    	END_IF;
    END_WHILE;
END_IF;
(* Rung 3 *)
IF P_On THEN AryByteTo(In := OUT[1], Size := 300, Order := _HIGH_LOW, OutVal := GBWORD); END_IF;
(* Rung 4 *)
IF P_On THEN
    unicode[0]:=16#4e00;
    unicode[1]:=16#4e01;
    unicode[2]:=16#4e03;
    unicode[3]:=16#4e07;
    unicode[4]:=16#4e08;
    unicode[5]:=16#4e09;
    unicode[6]:=16#4e0a;
    unicode[7]:=16#4e0b;
    unicode[8]:=16#4e0c;
    unicode[9]:=16#4e0d;
    unicode[10]:=16#4e0e;
    unicode[11]:=16#4e10;
    unicode[12]:=16#4e11;
    unicode[13]:=16#4e13;
    unicode[14]:=16#4e14;
    unicode[15]:=16#4e15;
    unicode[16]:=16#4e16;
    unicode[17]:=16#4e18;
    unicode[18]:=16#4e19;
    unicode[19]:=16#4e1a;
    unicode[20]:=16#4e1b;
    unicode[21]:=16#4e1c;
    unicode[22]:=16#4e1d;
    unicode[23]:=16#4e1e;
    unicode[24]:=16#4e22;
    unicode[25]:=16#4e24;
    unicode[26]:=16#4e25;
    unicode[27]:=16#4e27;
    unicode[28]:=16#4e28;
    unicode[29]:=16#4e2a;
    unicode[30]:=16#4e2b;
    unicode[31]:=16#4e2c;
    unicode[32]:=16#4e2d;
    unicode[33]:=16#4e30;
    unicode[34]:=16#4e32;
    unicode[35]:=16#4e34;
    unicode[36]:=16#4e36;
    unicode[37]:=16#4e38;
    unicode[38]:=16#4e39;
    unicode[39]:=16#4e3a;
    unicode[40]:=16#4e3b;
    unicode[41]:=16#4e3d;
    unicode[42]:=16#4e3e;
    unicode[43]:=16#4e3f;
    unicode[44]:=16#4e43;
    unicode[45]:=16#4e45;
    unicode[46]:=16#4e47;
    unicode[47]:=16#4e48;
    unicode[48]:=16#4e49;
    unicode[49]:=16#4e4b;
    unicode[50]:=16#4e4c;
    unicode[51]:=16#4e4d;
    unicode[52]:=16#4e4e;
    unicode[53]:=16#4e4f;
    unicode[54]:=16#4e50;
    unicode[55]:=16#4e52;
    unicode[56]:=16#4e53;
    unicode[57]:=16#4e54;
    unicode[58]:=16#4e56;
    unicode[59]:=16#4e58;
    unicode[60]:=16#4e59;
    unicode[61]:=16#4e5c;
    unicode[62]:=16#4e5d;
    unicode[63]:=16#4e5e;
    unicode[64]:=16#4e5f;
    unicode[65]:=16#4e60;
    unicode[66]:=16#4e61;
    unicode[67]:=16#4e66;
    unicode[68]:=16#4e69;
    unicode[69]:=16#4e70;
    unicode[70]:=16#4e71;
    unicode[71]:=16#4e73;
    unicode[72]:=16#4e7e;
    unicode[73]:=16#4e86;
    unicode[74]:=16#4e88;
    unicode[75]:=16#4e89;
    unicode[76]:=16#4e8b;
    unicode[77]:=16#4e8c;
    unicode[78]:=16#4e8d;
    unicode[79]:=16#4e8e;
    unicode[80]:=16#4e8f;
    unicode[81]:=16#4e91;
    unicode[82]:=16#4e92;
    unicode[83]:=16#4e93;
    unicode[84]:=16#4e94;
    unicode[85]:=16#4e95;
    unicode[86]:=16#4e98;
    unicode[87]:=16#4e9a;
    unicode[88]:=16#4e9b;
    unicode[89]:=16#4e9f;
    unicode[90]:=16#4ea0;
    unicode[91]:=16#4ea1;
    unicode[92]:=16#4ea2;
    unicode[93]:=16#4ea4;
    unicode[94]:=16#4ea5;
    unicode[95]:=16#4ea6;
    unicode[96]:=16#4ea7;
    unicode[97]:=16#4ea8;
    unicode[98]:=16#4ea9;
    unicode[99]:=16#4eab;
    unicode[100]:=16#4eac;
    unicode[101]:=16#4ead;
    unicode[102]:=16#4eae;
    unicode[103]:=16#4eb2;
    unicode[104]:=16#4eb3;
    unicode[105]:=16#4eb5;
    unicode[106]:=16#4eba;
    unicode[107]:=16#4ebb;
    unicode[108]:=16#4ebf;
    unicode[109]:=16#4ec0;
    unicode[110]:=16#4ec1;
    unicode[111]:=16#4ec2;
    unicode[112]:=16#4ec3;
    unicode[113]:=16#4ec4;
    unicode[114]:=16#4ec5;
    unicode[115]:=16#4ec6;
    unicode[116]:=16#4ec7;
    unicode[117]:=16#4ec9;
    unicode[118]:=16#4eca;
    unicode[119]:=16#4ecb;
    unicode[120]:=16#4ecd;
    unicode[121]:=16#4ece;
    unicode[122]:=16#4ed1;
    unicode[123]:=16#4ed3;
    unicode[124]:=16#4ed4;
    unicode[125]:=16#4ed5;
    unicode[126]:=16#4ed6;
    unicode[127]:=16#4ed7;
    unicode[128]:=16#4ed8;
    unicode[129]:=16#4ed9;
    unicode[130]:=16#4edd;
    unicode[131]:=16#4ede;
    unicode[132]:=16#4edf;
    unicode[133]:=16#4ee1;
    unicode[134]:=16#4ee3;
    unicode[135]:=16#4ee4;
    unicode[136]:=16#4ee5;
    unicode[137]:=16#4ee8;
    unicode[138]:=16#4eea;
    unicode[139]:=16#4eeb;
    unicode[140]:=16#4eec;
    unicode[141]:=16#4ef0;
    unicode[142]:=16#4ef2;
    unicode[143]:=16#4ef3;
    unicode[144]:=16#4ef5;
    unicode[145]:=16#4ef6;
    unicode[146]:=16#4ef7;
    unicode[147]:=16#4efb;
    unicode[148]:=16#4efd;
    unicode[149]:=16#4eff;
    unicode[150]:=16#4f01;
    unicode[151]:=16#4f09;
    unicode[152]:=16#4f0a;
    unicode[153]:=16#4f0d;
    unicode[154]:=16#4f0e;
    unicode[155]:=16#4f0f;
    unicode[156]:=16#4f10;
    unicode[157]:=16#4f11;
    unicode[158]:=16#4f17;
    unicode[159]:=16#4f18;
    unicode[160]:=16#4f19;
    unicode[161]:=16#4f1a;
    unicode[162]:=16#4f1b;
    unicode[163]:=16#4f1e;
    unicode[164]:=16#4f1f;
    unicode[165]:=16#4f20;
    unicode[166]:=16#4f22;
    unicode[167]:=16#4f24;
    unicode[168]:=16#4f25;
    unicode[169]:=16#4f26;
    unicode[170]:=16#4f27;
    unicode[171]:=16#4f2a;
    unicode[172]:=16#4f2b;
    unicode[173]:=16#4f2f;
    unicode[174]:=16#4f30;
    unicode[175]:=16#4f32;
    unicode[176]:=16#4f34;
    unicode[177]:=16#4f36;
    unicode[178]:=16#4f38;
    unicode[179]:=16#4f3a;
    unicode[180]:=16#4f3c;
    unicode[181]:=16#4f3d;
    unicode[182]:=16#4f43;
    unicode[183]:=16#4f46;
    unicode[184]:=16#4f4d;
    unicode[185]:=16#4f4e;
    unicode[186]:=16#4f4f;
    unicode[187]:=16#4f50;
    unicode[188]:=16#4f51;
    unicode[189]:=16#4f53;
    unicode[190]:=16#4f55;
    unicode[191]:=16#4f57;
    unicode[192]:=16#4f58;
    unicode[193]:=16#4f59;
    unicode[194]:=16#4f5a;
    unicode[195]:=16#4f5b;
    unicode[196]:=16#4f5c;
    unicode[197]:=16#4f5d;
    unicode[198]:=16#4f5e;
    unicode[199]:=16#4f5f;
    unicode[200]:=16#4f60;
    unicode[201]:=16#4f63;
    unicode[202]:=16#4f64;
    unicode[203]:=16#4f65;
    unicode[204]:=16#4f67;
    unicode[205]:=16#4f69;
    unicode[206]:=16#4f6c;
    unicode[207]:=16#4f6f;
    unicode[208]:=16#4f70;
    unicode[209]:=16#4f73;
    unicode[210]:=16#4f74;
    unicode[211]:=16#4f76;
    unicode[212]:=16#4f7b;
    unicode[213]:=16#4f7c;
    unicode[214]:=16#4f7e;
    unicode[215]:=16#4f7f;
    unicode[216]:=16#4f83;
    unicode[217]:=16#4f84;
    unicode[218]:=16#4f88;
    unicode[219]:=16#4f89;
    unicode[220]:=16#4f8b;
    unicode[221]:=16#4f8d;
    unicode[222]:=16#4f8f;
    unicode[223]:=16#4f91;
    unicode[224]:=16#4f94;
    unicode[225]:=16#4f97;
    unicode[226]:=16#4f9b;
    unicode[227]:=16#4f9d;
    unicode[228]:=16#4fa0;
    unicode[229]:=16#4fa3;
    unicode[230]:=16#4fa5;
    unicode[231]:=16#4fa6;
    unicode[232]:=16#4fa7;
    unicode[233]:=16#4fa8;
    unicode[234]:=16#4fa9;
    unicode[235]:=16#4faa;
    unicode[236]:=16#4fac;
    unicode[237]:=16#4fae;
    unicode[238]:=16#4faf;
    unicode[239]:=16#4fb5;
    unicode[240]:=16#4fbf;
    unicode[241]:=16#4fc3;
    unicode[242]:=16#4fc4;
    unicode[243]:=16#4fc5;
    unicode[244]:=16#4fca;
    unicode[245]:=16#4fce;
    unicode[246]:=16#4fcf;
    unicode[247]:=16#4fd0;
    unicode[248]:=16#4fd1;
    unicode[249]:=16#4fd7;
    unicode[250]:=16#4fd8;
    unicode[251]:=16#4fda;
    unicode[252]:=16#4fdc;
    unicode[253]:=16#4fdd;
    unicode[254]:=16#4fde;
    unicode[255]:=16#4fdf;
    unicode[256]:=16#4fe1;
    unicode[257]:=16#4fe3;
    unicode[258]:=16#4fe6;
    unicode[259]:=16#4fe8;
    unicode[260]:=16#4fe9;
    unicode[261]:=16#4fea;
    unicode[262]:=16#4fed;
    unicode[263]:=16#4fee;
    unicode[264]:=16#4fef;
    unicode[265]:=16#4ff1;
    unicode[266]:=16#4ff3;
    unicode[267]:=16#4ff8;
    unicode[268]:=16#4ffa;
    unicode[269]:=16#4ffe;
    unicode[270]:=16#500c;
    unicode[271]:=16#500d;
    unicode[272]:=16#500f;
    unicode[273]:=16#5012;
    unicode[274]:=16#5014;
    unicode[275]:=16#5018;
    unicode[276]:=16#5019;
    unicode[277]:=16#501a;
    unicode[278]:=16#501c;
    unicode[279]:=16#501f;
    unicode[280]:=16#5021;
    unicode[281]:=16#5025;
    unicode[282]:=16#5026;
    unicode[283]:=16#5028;
    unicode[284]:=16#5029;
    unicode[285]:=16#502a;
    unicode[286]:=16#502c;
    unicode[287]:=16#502d;
    unicode[288]:=16#502e;
    unicode[289]:=16#503a;
    unicode[290]:=16#503c;
    unicode[291]:=16#503e;
    unicode[292]:=16#5043;
    unicode[293]:=16#5047;
    unicode[294]:=16#5048;
    unicode[295]:=16#504c;
    unicode[296]:=16#504e;
    unicode[297]:=16#504f;
    unicode[298]:=16#5055;
    unicode[299]:=16#505a;
    unicode[300]:=16#505c;
    unicode[301]:=16#5065;
    unicode[302]:=16#506c;
    unicode[303]:=16#5076;
    unicode[304]:=16#5077;
    unicode[305]:=16#507b;
    unicode[306]:=16#507e;
    unicode[307]:=16#507f;
    unicode[308]:=16#5080;
    unicode[309]:=16#5085;
    unicode[310]:=16#5088;
    unicode[311]:=16#508d;
    unicode[312]:=16#50a3;
    unicode[313]:=16#50a5;
    unicode[314]:=16#50a7;
    unicode[315]:=16#50a8;
    unicode[316]:=16#50a9;
    unicode[317]:=16#50ac;
    unicode[318]:=16#50b2;
    unicode[319]:=16#50ba;
    unicode[320]:=16#50bb;
    unicode[321]:=16#50cf;
    unicode[322]:=16#50d6;
    unicode[323]:=16#50da;
    unicode[324]:=16#50e6;
    unicode[325]:=16#50e7;
    unicode[326]:=16#50ec;
    unicode[327]:=16#50ed;
    unicode[328]:=16#50ee;
    unicode[329]:=16#50f3;
    unicode[330]:=16#50f5;
    unicode[331]:=16#50fb;
    unicode[332]:=16#5106;
    unicode[333]:=16#5107;
    unicode[334]:=16#510b;
    unicode[335]:=16#5112;
    unicode[336]:=16#5121;
    unicode[337]:=16#513f;
    unicode[338]:=16#5140;
    unicode[339]:=16#5141;
    unicode[340]:=16#5143;
    unicode[341]:=16#5144;
    unicode[342]:=16#5145;
    unicode[343]:=16#5146;
    unicode[344]:=16#5148;
    unicode[345]:=16#5149;
    unicode[346]:=16#514b;
    unicode[347]:=16#514d;
    unicode[348]:=16#5151;
    unicode[349]:=16#5154;
    unicode[350]:=16#5155;
    unicode[351]:=16#5156;
    unicode[352]:=16#515a;
    unicode[353]:=16#515c;
    unicode[354]:=16#5162;
    unicode[355]:=16#5165;
    unicode[356]:=16#5168;
    unicode[357]:=16#516b;
    unicode[358]:=16#516c;
    unicode[359]:=16#516d;
    unicode[360]:=16#516e;
    unicode[361]:=16#5170;
    unicode[362]:=16#5171;
    unicode[363]:=16#5173;
    unicode[364]:=16#5174;
    unicode[365]:=16#5175;
    unicode[366]:=16#5176;
    unicode[367]:=16#5177;
    unicode[368]:=16#5178;
    unicode[369]:=16#5179;
    unicode[370]:=16#517b;
    unicode[371]:=16#517c;
    unicode[372]:=16#517d;
    unicode[373]:=16#5180;
    unicode[374]:=16#5181;
    unicode[375]:=16#5182;
    unicode[376]:=16#5185;
    unicode[377]:=16#5188;
    unicode[378]:=16#5189;
    unicode[379]:=16#518c;
    unicode[380]:=16#518d;
    unicode[381]:=16#5192;
    unicode[382]:=16#5195;
    unicode[383]:=16#5196;
    unicode[384]:=16#5197;
    unicode[385]:=16#5199;
    unicode[386]:=16#519b;
    unicode[387]:=16#519c;
    unicode[388]:=16#51a0;
    unicode[389]:=16#51a2;
    unicode[390]:=16#51a4;
    unicode[391]:=16#51a5;
    unicode[392]:=16#51ab;
    unicode[393]:=16#51ac;
    unicode[394]:=16#51af;
    unicode[395]:=16#51b0;
    unicode[396]:=16#51b1;
    unicode[397]:=16#51b2;
    unicode[398]:=16#51b3;
    unicode[399]:=16#51b5;
    unicode[400]:=16#51b6;
    unicode[401]:=16#51b7;
    unicode[402]:=16#51bb;
    unicode[403]:=16#51bc;
    unicode[404]:=16#51bd;
    unicode[405]:=16#51c0;
    unicode[406]:=16#51c4;
    unicode[407]:=16#51c6;
    unicode[408]:=16#51c7;
    unicode[409]:=16#51c9;
    unicode[410]:=16#51cb;
    unicode[411]:=16#51cc;
    unicode[412]:=16#51cf;
    unicode[413]:=16#51d1;
    unicode[414]:=16#51db;
    unicode[415]:=16#51dd;
    unicode[416]:=16#51e0;
    unicode[417]:=16#51e1;
    unicode[418]:=16#51e4;
    unicode[419]:=16#51eb;
    unicode[420]:=16#51ed;
    unicode[421]:=16#51ef;
    unicode[422]:=16#51f0;
    unicode[423]:=16#51f3;
    unicode[424]:=16#51f5;
    unicode[425]:=16#51f6;
    unicode[426]:=16#51f8;
    unicode[427]:=16#51f9;
    unicode[428]:=16#51fa;
    unicode[429]:=16#51fb;
    unicode[430]:=16#51fc;
    unicode[431]:=16#51fd;
    unicode[432]:=16#51ff;
    unicode[433]:=16#5200;
    unicode[434]:=16#5201;
    unicode[435]:=16#5202;
    unicode[436]:=16#5203;
    unicode[437]:=16#5206;
    unicode[438]:=16#5207;
    unicode[439]:=16#5208;
    unicode[440]:=16#520a;
    unicode[441]:=16#520d;
    unicode[442]:=16#520e;
    unicode[443]:=16#5211;
    unicode[444]:=16#5212;
    unicode[445]:=16#5216;
    unicode[446]:=16#5217;
    unicode[447]:=16#5218;
    unicode[448]:=16#5219;
    unicode[449]:=16#521a;
    unicode[450]:=16#521b;
    unicode[451]:=16#521d;
    unicode[452]:=16#5220;
    unicode[453]:=16#5224;
    unicode[454]:=16#5228;
    unicode[455]:=16#5229;
    unicode[456]:=16#522b;
    unicode[457]:=16#522d;
    unicode[458]:=16#522e;
    unicode[459]:=16#5230;
    unicode[460]:=16#5233;
    unicode[461]:=16#5236;
    unicode[462]:=16#5237;
    unicode[463]:=16#5238;
    unicode[464]:=16#5239;
    unicode[465]:=16#523a;
    unicode[466]:=16#523b;
    unicode[467]:=16#523d;
    unicode[468]:=16#523f;
    unicode[469]:=16#5240;
    unicode[470]:=16#5241;
    unicode[471]:=16#5242;
    unicode[472]:=16#5243;
    unicode[473]:=16#524a;
    unicode[474]:=16#524c;
    unicode[475]:=16#524d;
    unicode[476]:=16#5250;
    unicode[477]:=16#5251;
    unicode[478]:=16#5254;
    unicode[479]:=16#5256;
    unicode[480]:=16#525c;
    unicode[481]:=16#525e;
    unicode[482]:=16#5261;
    unicode[483]:=16#5265;
    unicode[484]:=16#5267;
    unicode[485]:=16#5269;
    unicode[486]:=16#526a;
    unicode[487]:=16#526f;
    unicode[488]:=16#5272;
    unicode[489]:=16#527d;
    unicode[490]:=16#527f;
    unicode[491]:=16#5281;
    unicode[492]:=16#5282;
    unicode[493]:=16#5288;
    unicode[494]:=16#5290;
    unicode[495]:=16#5293;
    unicode[496]:=16#529b;
    unicode[497]:=16#529d;
    unicode[498]:=16#529e;
    unicode[499]:=16#529f;
    unicode[500]:=16#52a0;
    unicode[501]:=16#52a1;
    unicode[502]:=16#52a2;
    unicode[503]:=16#52a3;
    unicode[504]:=16#52a8;
    unicode[505]:=16#52a9;
    unicode[506]:=16#52aa;
    unicode[507]:=16#52ab;
    unicode[508]:=16#52ac;
    unicode[509]:=16#52ad;
    unicode[510]:=16#52b1;
    unicode[511]:=16#52b2;
    unicode[512]:=16#52b3;
    unicode[513]:=16#52be;
    unicode[514]:=16#52bf;
    unicode[515]:=16#52c3;
    unicode[516]:=16#52c7;
    unicode[517]:=16#52c9;
    unicode[518]:=16#52cb;
    unicode[519]:=16#52d0;
    unicode[520]:=16#52d2;
    unicode[521]:=16#52d6;
    unicode[522]:=16#52d8;
    unicode[523]:=16#52df;
    unicode[524]:=16#52e4;
    unicode[525]:=16#52f0;
    unicode[526]:=16#52f9;
    unicode[527]:=16#52fa;
    unicode[528]:=16#52fe;
    unicode[529]:=16#52ff;
    unicode[530]:=16#5300;
    unicode[531]:=16#5305;
    unicode[532]:=16#5306;
    unicode[533]:=16#5308;
    unicode[534]:=16#530d;
    unicode[535]:=16#530f;
    unicode[536]:=16#5310;
    unicode[537]:=16#5315;
    unicode[538]:=16#5316;
    unicode[539]:=16#5317;
    unicode[540]:=16#5319;
    unicode[541]:=16#531a;
    unicode[542]:=16#531d;
    unicode[543]:=16#5320;
    unicode[544]:=16#5321;
    unicode[545]:=16#5323;
    unicode[546]:=16#5326;
    unicode[547]:=16#532a;
    unicode[548]:=16#532e;
    unicode[549]:=16#5339;
    unicode[550]:=16#533a;
    unicode[551]:=16#533b;
    unicode[552]:=16#533e;
    unicode[553]:=16#533f;
    unicode[554]:=16#5341;
    unicode[555]:=16#5343;
    unicode[556]:=16#5345;
    unicode[557]:=16#5347;
    unicode[558]:=16#5348;
    unicode[559]:=16#5349;
    unicode[560]:=16#534a;
    unicode[561]:=16#534e;
    unicode[562]:=16#534f;
    unicode[563]:=16#5351;
    unicode[564]:=16#5352;
    unicode[565]:=16#5353;
    unicode[566]:=16#5355;
    unicode[567]:=16#5356;
    unicode[568]:=16#5357;
    unicode[569]:=16#535a;
    unicode[570]:=16#535c;
    unicode[571]:=16#535e;
    unicode[572]:=16#535f;
    unicode[573]:=16#5360;
    unicode[574]:=16#5361;
    unicode[575]:=16#5362;
    unicode[576]:=16#5363;
    unicode[577]:=16#5364;
    unicode[578]:=16#5366;
    unicode[579]:=16#5367;
    unicode[580]:=16#5369;
    unicode[581]:=16#536b;
    unicode[582]:=16#536e;
    unicode[583]:=16#536f;
    unicode[584]:=16#5370;
    unicode[585]:=16#5371;
    unicode[586]:=16#5373;
    unicode[587]:=16#5374;
    unicode[588]:=16#5375;
    unicode[589]:=16#5377;
    unicode[590]:=16#5378;
    unicode[591]:=16#537a;
    unicode[592]:=16#537f;
    unicode[593]:=16#5382;
    unicode[594]:=16#5384;
    unicode[595]:=16#5385;
    unicode[596]:=16#5386;
    unicode[597]:=16#5389;
    unicode[598]:=16#538b;
    unicode[599]:=16#538c;
    unicode[600]:=16#538d;
    unicode[601]:=16#5395;
    unicode[602]:=16#5398;
    unicode[603]:=16#539a;
    unicode[604]:=16#539d;
    unicode[605]:=16#539f;
    unicode[606]:=16#53a2;
    unicode[607]:=16#53a3;
    unicode[608]:=16#53a5;
    unicode[609]:=16#53a6;
    unicode[610]:=16#53a8;
    unicode[611]:=16#53a9;
    unicode[612]:=16#53ae;
    unicode[613]:=16#53b6;
    unicode[614]:=16#53bb;
    unicode[615]:=16#53bf;
    unicode[616]:=16#53c1;
    unicode[617]:=16#53c2;
    unicode[618]:=16#53c8;
    unicode[619]:=16#53c9;
    unicode[620]:=16#53ca;
    unicode[621]:=16#53cb;
    unicode[622]:=16#53cc;
    unicode[623]:=16#53cd;
    unicode[624]:=16#53d1;
    unicode[625]:=16#53d4;
    unicode[626]:=16#53d6;
    unicode[627]:=16#53d7;
    unicode[628]:=16#53d8;
    unicode[629]:=16#53d9;
    unicode[630]:=16#53db;
    unicode[631]:=16#53df;
    unicode[632]:=16#53e0;
    unicode[633]:=16#53e3;
    unicode[634]:=16#53e4;
    unicode[635]:=16#53e5;
    unicode[636]:=16#53e6;
    unicode[637]:=16#53e8;
    unicode[638]:=16#53e9;
    unicode[639]:=16#53ea;
    unicode[640]:=16#53eb;
    unicode[641]:=16#53ec;
    unicode[642]:=16#53ed;
    unicode[643]:=16#53ee;
    unicode[644]:=16#53ef;
    unicode[645]:=16#53f0;
    unicode[646]:=16#53f1;
    unicode[647]:=16#53f2;
    unicode[648]:=16#53f3;
    unicode[649]:=16#53f5;
    unicode[650]:=16#53f6;
    unicode[651]:=16#53f7;
    unicode[652]:=16#53f8;
    unicode[653]:=16#53f9;
    unicode[654]:=16#53fb;
    unicode[655]:=16#53fc;
    unicode[656]:=16#53fd;
    unicode[657]:=16#5401;
    unicode[658]:=16#5403;
    unicode[659]:=16#5404;
    unicode[660]:=16#5406;
    unicode[661]:=16#5408;
    unicode[662]:=16#5409;
    unicode[663]:=16#540a;
    unicode[664]:=16#540c;
    unicode[665]:=16#540d;
    unicode[666]:=16#540e;
    unicode[667]:=16#540f;
    unicode[668]:=16#5410;
    unicode[669]:=16#5411;
    unicode[670]:=16#5412;
    unicode[671]:=16#5413;
    unicode[672]:=16#5415;
    unicode[673]:=16#5416;
    unicode[674]:=16#5417;
    unicode[675]:=16#541b;
    unicode[676]:=16#541d;
    unicode[677]:=16#541e;
    unicode[678]:=16#541f;
    unicode[679]:=16#5420;
    unicode[680]:=16#5421;
    unicode[681]:=16#5423;
    unicode[682]:=16#5426;
    unicode[683]:=16#5427;
    unicode[684]:=16#5428;
    unicode[685]:=16#5429;
    unicode[686]:=16#542b;
    unicode[687]:=16#542c;
    unicode[688]:=16#542d;
    unicode[689]:=16#542e;
    unicode[690]:=16#542f;
    unicode[691]:=16#5431;
    unicode[692]:=16#5432;
    unicode[693]:=16#5434;
    unicode[694]:=16#5435;
    unicode[695]:=16#5438;
    unicode[696]:=16#5439;
    unicode[697]:=16#543b;
    unicode[698]:=16#543c;
    unicode[699]:=16#543e;
    unicode[700]:=16#5440;
    unicode[701]:=16#5443;
    unicode[702]:=16#5446;
    unicode[703]:=16#5448;
    unicode[704]:=16#544a;
    unicode[705]:=16#544b;
    unicode[706]:=16#5450;
    unicode[707]:=16#5452;
    unicode[708]:=16#5453;
    unicode[709]:=16#5454;
    unicode[710]:=16#5455;
    unicode[711]:=16#5456;
    unicode[712]:=16#5457;
    unicode[713]:=16#5458;
    unicode[714]:=16#5459;
    unicode[715]:=16#545b;
    unicode[716]:=16#545c;
    unicode[717]:=16#5462;
    unicode[718]:=16#5464;
    unicode[719]:=16#5466;
    unicode[720]:=16#5468;
    unicode[721]:=16#5471;
    unicode[722]:=16#5472;
    unicode[723]:=16#5473;
    unicode[724]:=16#5475;
    unicode[725]:=16#5476;
    unicode[726]:=16#5477;
    unicode[727]:=16#5478;
    unicode[728]:=16#547b;
    unicode[729]:=16#547c;
    unicode[730]:=16#547d;
    unicode[731]:=16#5480;
    unicode[732]:=16#5482;
    unicode[733]:=16#5484;
    unicode[734]:=16#5486;
    unicode[735]:=16#548b;
    unicode[736]:=16#548c;
    unicode[737]:=16#548e;
    unicode[738]:=16#548f;
    unicode[739]:=16#5490;
    unicode[740]:=16#5492;
    unicode[741]:=16#5494;
    unicode[742]:=16#5495;
    unicode[743]:=16#5496;
    unicode[744]:=16#5499;
    unicode[745]:=16#549a;
    unicode[746]:=16#549b;
    unicode[747]:=16#549d;
    unicode[748]:=16#54a3;
    unicode[749]:=16#54a4;
    unicode[750]:=16#54a6;
    unicode[751]:=16#54a7;
    unicode[752]:=16#54a8;
    unicode[753]:=16#54a9;
    unicode[754]:=16#54aa;
    unicode[755]:=16#54ab;
    unicode[756]:=16#54ac;
    unicode[757]:=16#54ad;
    unicode[758]:=16#54af;
    unicode[759]:=16#54b1;
    unicode[760]:=16#54b3;
    unicode[761]:=16#54b4;
    unicode[762]:=16#54b8;
    unicode[763]:=16#54bb;
    unicode[764]:=16#54bd;
    unicode[765]:=16#54bf;
    unicode[766]:=16#54c0;
    unicode[767]:=16#54c1;
    unicode[768]:=16#54c2;
    unicode[769]:=16#54c4;
    unicode[770]:=16#54c6;
    unicode[771]:=16#54c7;
    unicode[772]:=16#54c8;
    unicode[773]:=16#54c9;
    unicode[774]:=16#54cc;
    unicode[775]:=16#54cd;
    unicode[776]:=16#54ce;
    unicode[777]:=16#54cf;
    unicode[778]:=16#54d0;
    unicode[779]:=16#54d1;
    unicode[780]:=16#54d2;
    unicode[781]:=16#54d3;
    unicode[782]:=16#54d4;
    unicode[783]:=16#54d5;
    unicode[784]:=16#54d7;
    unicode[785]:=16#54d9;
    unicode[786]:=16#54da;
    unicode[787]:=16#54dc;
    unicode[788]:=16#54dd;
    unicode[789]:=16#54de;
    unicode[790]:=16#54df;
    unicode[791]:=16#54e5;
    unicode[792]:=16#54e6;
    unicode[793]:=16#54e7;
    unicode[794]:=16#54e8;
    unicode[795]:=16#54e9;
    unicode[796]:=16#54ea;
    unicode[797]:=16#54ed;
    unicode[798]:=16#54ee;
    unicode[799]:=16#54f2;
    unicode[800]:=16#54f3;
    unicode[801]:=16#54fa;
    unicode[802]:=16#54fc;
    unicode[803]:=16#54fd;
    unicode[804]:=16#54ff;
    unicode[805]:=16#5501;
    unicode[806]:=16#5506;
    unicode[807]:=16#5507;
    unicode[808]:=16#5509;
    unicode[809]:=16#550f;
    unicode[810]:=16#5510;
    unicode[811]:=16#5511;
    unicode[812]:=16#5514;
    unicode[813]:=16#551b;
    unicode[814]:=16#5520;
    unicode[815]:=16#5522;
    unicode[816]:=16#5523;
    unicode[817]:=16#5524;
    unicode[818]:=16#5527;
    unicode[819]:=16#552a;
    unicode[820]:=16#552c;
    unicode[821]:=16#552e;
    unicode[822]:=16#552f;
    unicode[823]:=16#5530;
    unicode[824]:=16#5531;
    unicode[825]:=16#5533;
    unicode[826]:=16#5537;
    unicode[827]:=16#553c;
    unicode[828]:=16#553e;
    unicode[829]:=16#553f;
    unicode[830]:=16#5541;
    unicode[831]:=16#5543;
    unicode[832]:=16#5544;
    unicode[833]:=16#5546;
    unicode[834]:=16#5549;
    unicode[835]:=16#554a;
    unicode[836]:=16#5550;
    unicode[837]:=16#5555;
    unicode[838]:=16#5556;
    unicode[839]:=16#555c;
    unicode[840]:=16#5561;
    unicode[841]:=16#5564;
    unicode[842]:=16#5565;
    unicode[843]:=16#5566;
    unicode[844]:=16#5567;
    unicode[845]:=16#556a;
    unicode[846]:=16#556c;
    unicode[847]:=16#556d;
    unicode[848]:=16#556e;
    unicode[849]:=16#5575;
    unicode[850]:=16#5576;
    unicode[851]:=16#5577;
    unicode[852]:=16#5578;
    unicode[853]:=16#557b;
    unicode[854]:=16#557c;
    unicode[855]:=16#557e;
    unicode[856]:=16#5580;
    unicode[857]:=16#5581;
    unicode[858]:=16#5582;
    unicode[859]:=16#5583;
    unicode[860]:=16#5584;
    unicode[861]:=16#5587;
    unicode[862]:=16#5588;
    unicode[863]:=16#5589;
    unicode[864]:=16#558a;
    unicode[865]:=16#558b;
    unicode[866]:=16#558f;
    unicode[867]:=16#5591;
    unicode[868]:=16#5594;
    unicode[869]:=16#5598;
    unicode[870]:=16#5599;
    unicode[871]:=16#559c;
    unicode[872]:=16#559d;
    unicode[873]:=16#559f;
    unicode[874]:=16#55a7;
    unicode[875]:=16#55b1;
    unicode[876]:=16#55b3;
    unicode[877]:=16#55b5;
    unicode[878]:=16#55b7;
    unicode[879]:=16#55b9;
    unicode[880]:=16#55bb;
    unicode[881]:=16#55bd;
    unicode[882]:=16#55be;
    unicode[883]:=16#55c4;
    unicode[884]:=16#55c5;
    unicode[885]:=16#55c9;
    unicode[886]:=16#55cc;
    unicode[887]:=16#55cd;
    unicode[888]:=16#55d1;
    unicode[889]:=16#55d2;
    unicode[890]:=16#55d3;
    unicode[891]:=16#55d4;
    unicode[892]:=16#55d6;
    unicode[893]:=16#55dc;
    unicode[894]:=16#55dd;
    unicode[895]:=16#55df;
    unicode[896]:=16#55e1;
    unicode[897]:=16#55e3;
    unicode[898]:=16#55e4;
    unicode[899]:=16#55e5;
    unicode[900]:=16#55e6;
    unicode[901]:=16#55e8;
    unicode[902]:=16#55ea;
    unicode[903]:=16#55eb;
    unicode[904]:=16#55ec;
    unicode[905]:=16#55ef;
    unicode[906]:=16#55f2;
    unicode[907]:=16#55f3;
    unicode[908]:=16#55f5;
    unicode[909]:=16#55f7;
    unicode[910]:=16#55fd;
    unicode[911]:=16#55fe;
    unicode[912]:=16#5600;
    unicode[913]:=16#5601;
    unicode[914]:=16#5608;
    unicode[915]:=16#5609;
    unicode[916]:=16#560c;
    unicode[917]:=16#560e;
    unicode[918]:=16#560f;
    unicode[919]:=16#5618;
    unicode[920]:=16#561b;
    unicode[921]:=16#561e;
    unicode[922]:=16#561f;
    unicode[923]:=16#5623;
    unicode[924]:=16#5624;
    unicode[925]:=16#5627;
    unicode[926]:=16#562c;
    unicode[927]:=16#562d;
    unicode[928]:=16#5631;
    unicode[929]:=16#5632;
    unicode[930]:=16#5634;
    unicode[931]:=16#5636;
    unicode[932]:=16#5639;
    unicode[933]:=16#563b;
    unicode[934]:=16#563f;
    unicode[935]:=16#564c;
    unicode[936]:=16#564d;
    unicode[937]:=16#564e;
    unicode[938]:=16#5654;
    unicode[939]:=16#5657;
    unicode[940]:=16#5658;
    unicode[941]:=16#5659;
    unicode[942]:=16#565c;
    unicode[943]:=16#5662;
    unicode[944]:=16#5664;
    unicode[945]:=16#5668;
    unicode[946]:=16#5669;
    unicode[947]:=16#566a;
    unicode[948]:=16#566b;
    unicode[949]:=16#566c;
    unicode[950]:=16#5671;
    unicode[951]:=16#5676;
    unicode[952]:=16#567b;
    unicode[953]:=16#567c;
    unicode[954]:=16#5685;
    unicode[955]:=16#5686;
    unicode[956]:=16#568e;
    unicode[957]:=16#568f;
    unicode[958]:=16#5693;
    unicode[959]:=16#56a3;
    unicode[960]:=16#56af;
    unicode[961]:=16#56b7;
    unicode[962]:=16#56bc;
    unicode[963]:=16#56ca;
    unicode[964]:=16#56d4;
    unicode[965]:=16#56d7;
    unicode[966]:=16#56da;
    unicode[967]:=16#56db;
    unicode[968]:=16#56dd;
    unicode[969]:=16#56de;
    unicode[970]:=16#56df;
    unicode[971]:=16#56e0;
    unicode[972]:=16#56e1;
    unicode[973]:=16#56e2;
    unicode[974]:=16#56e4;
    unicode[975]:=16#56eb;
    unicode[976]:=16#56ed;
    unicode[977]:=16#56f0;
    unicode[978]:=16#56f1;
    unicode[979]:=16#56f4;
    unicode[980]:=16#56f5;
    unicode[981]:=16#56f9;
    unicode[982]:=16#56fa;
    unicode[983]:=16#56fd;
    unicode[984]:=16#56fe;
    unicode[985]:=16#56ff;
    unicode[986]:=16#5703;
    unicode[987]:=16#5704;
    unicode[988]:=16#5706;
    unicode[989]:=16#5708;
    unicode[990]:=16#5709;
    unicode[991]:=16#570a;
    unicode[992]:=16#571c;
    unicode[993]:=16#571f;
    unicode[994]:=16#5723;
    unicode[995]:=16#5728;
    unicode[996]:=16#5729;
    unicode[997]:=16#572a;
    unicode[998]:=16#572c;
    unicode[999]:=16#572d;           //unicode码 0-999
END_IF;

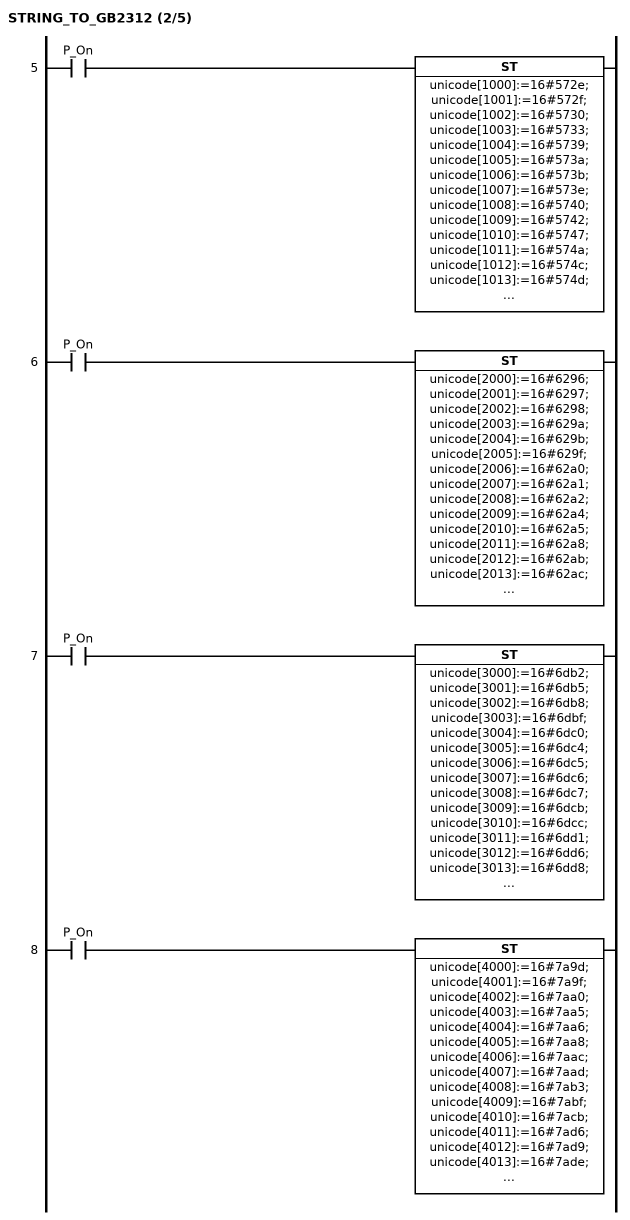
(* [picture p2: STRING_TO_GB2312, rungs 5-8] *)
(* Rung 5 *)
IF P_On THEN
    unicode[1000]:=16#572e;
    unicode[1001]:=16#572f;
    unicode[1002]:=16#5730;
    unicode[1003]:=16#5733;
    unicode[1004]:=16#5739;
    unicode[1005]:=16#573a;
    unicode[1006]:=16#573b;
    unicode[1007]:=16#573e;
    unicode[1008]:=16#5740;
    unicode[1009]:=16#5742;
    unicode[1010]:=16#5747;
    unicode[1011]:=16#574a;
    unicode[1012]:=16#574c;
    unicode[1013]:=16#574d;
    unicode[1014]:=16#574e;
    unicode[1015]:=16#574f;
    unicode[1016]:=16#5750;
    unicode[1017]:=16#5751;
    unicode[1018]:=16#5757;
    unicode[1019]:=16#575a;
    unicode[1020]:=16#575b;
    unicode[1021]:=16#575c;
    unicode[1022]:=16#575d;
    unicode[1023]:=16#575e;
    unicode[1024]:=16#575f;
    unicode[1025]:=16#5760;
    unicode[1026]:=16#5761;
    unicode[1027]:=16#5764;
    unicode[1028]:=16#5766;
    unicode[1029]:=16#5768;
    unicode[1030]:=16#5769;
    unicode[1031]:=16#576a;
    unicode[1032]:=16#576b;
    unicode[1033]:=16#576d;
    unicode[1034]:=16#576f;
    unicode[1035]:=16#5773;
    unicode[1036]:=16#5776;
    unicode[1037]:=16#5777;
    unicode[1038]:=16#577b;
    unicode[1039]:=16#577c;
    unicode[1040]:=16#5782;
    unicode[1041]:=16#5783;
    unicode[1042]:=16#5784;
    unicode[1043]:=16#5785;
    unicode[1044]:=16#5786;
    unicode[1045]:=16#578b;
    unicode[1046]:=16#578c;
    unicode[1047]:=16#5792;
    unicode[1048]:=16#5793;
    unicode[1049]:=16#579b;
    unicode[1050]:=16#57a0;
    unicode[1051]:=16#57a1;
    unicode[1052]:=16#57a2;
    unicode[1053]:=16#57a3;
    unicode[1054]:=16#57a4;
    unicode[1055]:=16#57a6;
    unicode[1056]:=16#57a7;
    unicode[1057]:=16#57a9;
    unicode[1058]:=16#57ab;
    unicode[1059]:=16#57ad;
    unicode[1060]:=16#57ae;
    unicode[1061]:=16#57b2;
    unicode[1062]:=16#57b4;
    unicode[1063]:=16#57b8;
    unicode[1064]:=16#57c2;
    unicode[1065]:=16#57c3;
    unicode[1066]:=16#57cb;
    unicode[1067]:=16#57ce;
    unicode[1068]:=16#57cf;
    unicode[1069]:=16#57d2;
    unicode[1070]:=16#57d4;
    unicode[1071]:=16#57d5;
    unicode[1072]:=16#57d8;
    unicode[1073]:=16#57d9;
    unicode[1074]:=16#57da;
    unicode[1075]:=16#57dd;
    unicode[1076]:=16#57df;
    unicode[1077]:=16#57e0;
    unicode[1078]:=16#57e4;
    unicode[1079]:=16#57ed;
    unicode[1080]:=16#57ef;
    unicode[1081]:=16#57f4;
    unicode[1082]:=16#57f8;
    unicode[1083]:=16#57f9;
    unicode[1084]:=16#57fa;
    unicode[1085]:=16#57fd;
    unicode[1086]:=16#5800;
    unicode[1087]:=16#5802;
    unicode[1088]:=16#5806;
    unicode[1089]:=16#5807;
    unicode[1090]:=16#580b;
    unicode[1091]:=16#580d;
    unicode[1092]:=16#5811;
    unicode[1093]:=16#5815;
    unicode[1094]:=16#5819;
    unicode[1095]:=16#581e;
    unicode[1096]:=16#5820;
    unicode[1097]:=16#5821;
    unicode[1098]:=16#5824;
    unicode[1099]:=16#582a;
    unicode[1100]:=16#5830;
    unicode[1101]:=16#5835;
    unicode[1102]:=16#5844;
    unicode[1103]:=16#584c;
    unicode[1104]:=16#584d;
    unicode[1105]:=16#5851;
    unicode[1106]:=16#5854;
    unicode[1107]:=16#5858;
    unicode[1108]:=16#585e;
    unicode[1109]:=16#5865;
    unicode[1110]:=16#586b;
    unicode[1111]:=16#586c;
    unicode[1112]:=16#587e;
    unicode[1113]:=16#5880;
    unicode[1114]:=16#5881;
    unicode[1115]:=16#5883;
    unicode[1116]:=16#5885;
    unicode[1117]:=16#5889;
    unicode[1118]:=16#5892;
    unicode[1119]:=16#5893;
    unicode[1120]:=16#5899;
    unicode[1121]:=16#589a;
    unicode[1122]:=16#589e;
    unicode[1123]:=16#589f;
    unicode[1124]:=16#58a8;
    unicode[1125]:=16#58a9;
    unicode[1126]:=16#58bc;
    unicode[1127]:=16#58c1;
    unicode[1128]:=16#58c5;
    unicode[1129]:=16#58d1;
    unicode[1130]:=16#58d5;
    unicode[1131]:=16#58e4;
    unicode[1132]:=16#58eb;
    unicode[1133]:=16#58ec;
    unicode[1134]:=16#58ee;
    unicode[1135]:=16#58f0;
    unicode[1136]:=16#58f3;
    unicode[1137]:=16#58f6;
    unicode[1138]:=16#58f9;
    unicode[1139]:=16#5902;
    unicode[1140]:=16#5904;
    unicode[1141]:=16#5907;
    unicode[1142]:=16#590d;
    unicode[1143]:=16#590f;
    unicode[1144]:=16#5914;
    unicode[1145]:=16#5915;
    unicode[1146]:=16#5916;
    unicode[1147]:=16#5919;
    unicode[1148]:=16#591a;
    unicode[1149]:=16#591c;
    unicode[1150]:=16#591f;
    unicode[1151]:=16#5924;
    unicode[1152]:=16#5925;
    unicode[1153]:=16#5927;
    unicode[1154]:=16#5929;
    unicode[1155]:=16#592a;
    unicode[1156]:=16#592b;
    unicode[1157]:=16#592d;
    unicode[1158]:=16#592e;
    unicode[1159]:=16#592f;
    unicode[1160]:=16#5931;
    unicode[1161]:=16#5934;
    unicode[1162]:=16#5937;
    unicode[1163]:=16#5938;
    unicode[1164]:=16#5939;
    unicode[1165]:=16#593a;
    unicode[1166]:=16#593c;
    unicode[1167]:=16#5941;
    unicode[1168]:=16#5942;
    unicode[1169]:=16#5944;
    unicode[1170]:=16#5947;
    unicode[1171]:=16#5948;
    unicode[1172]:=16#5949;
    unicode[1173]:=16#594b;
    unicode[1174]:=16#594e;
    unicode[1175]:=16#594f;
    unicode[1176]:=16#5951;
    unicode[1177]:=16#5954;
    unicode[1178]:=16#5955;
    unicode[1179]:=16#5956;
    unicode[1180]:=16#5957;
    unicode[1181]:=16#5958;
    unicode[1182]:=16#595a;
    unicode[1183]:=16#5960;
    unicode[1184]:=16#5962;
    unicode[1185]:=16#5965;
    unicode[1186]:=16#5973;
    unicode[1187]:=16#5974;
    unicode[1188]:=16#5976;
    unicode[1189]:=16#5978;
    unicode[1190]:=16#5979;
    unicode[1191]:=16#597d;
    unicode[1192]:=16#5981;
    unicode[1193]:=16#5982;
    unicode[1194]:=16#5983;
    unicode[1195]:=16#5984;
    unicode[1196]:=16#5986;
    unicode[1197]:=16#5987;
    unicode[1198]:=16#5988;
    unicode[1199]:=16#598a;
    unicode[1200]:=16#598d;
    unicode[1201]:=16#5992;
    unicode[1202]:=16#5993;
    unicode[1203]:=16#5996;
    unicode[1204]:=16#5997;
    unicode[1205]:=16#5999;
    unicode[1206]:=16#599e;
    unicode[1207]:=16#59a3;
    unicode[1208]:=16#59a4;
    unicode[1209]:=16#59a5;
    unicode[1210]:=16#59a8;
    unicode[1211]:=16#59a9;
    unicode[1212]:=16#59aa;
    unicode[1213]:=16#59ab;
    unicode[1214]:=16#59ae;
    unicode[1215]:=16#59af;
    unicode[1216]:=16#59b2;
    unicode[1217]:=16#59b9;
    unicode[1218]:=16#59bb;
    unicode[1219]:=16#59be;
    unicode[1220]:=16#59c6;
    unicode[1221]:=16#59ca;
    unicode[1222]:=16#59cb;
    unicode[1223]:=16#59d0;
    unicode[1224]:=16#59d1;
    unicode[1225]:=16#59d2;
    unicode[1226]:=16#59d3;
    unicode[1227]:=16#59d4;
    unicode[1228]:=16#59d7;
    unicode[1229]:=16#59d8;
    unicode[1230]:=16#59da;
    unicode[1231]:=16#59dc;
    unicode[1232]:=16#59dd;
    unicode[1233]:=16#59e3;
    unicode[1234]:=16#59e5;
    unicode[1235]:=16#59e8;
    unicode[1236]:=16#59ec;
    unicode[1237]:=16#59f9;
    unicode[1238]:=16#59fb;
    unicode[1239]:=16#59ff;
    unicode[1240]:=16#5a01;
    unicode[1241]:=16#5a03;
    unicode[1242]:=16#5a04;
    unicode[1243]:=16#5a05;
    unicode[1244]:=16#5a06;
    unicode[1245]:=16#5a07;
    unicode[1246]:=16#5a08;
    unicode[1247]:=16#5a09;
    unicode[1248]:=16#5a0c;
    unicode[1249]:=16#5a11;
    unicode[1250]:=16#5a13;
    unicode[1251]:=16#5a18;
    unicode[1252]:=16#5a1c;
    unicode[1253]:=16#5a1f;
    unicode[1254]:=16#5a20;
    unicode[1255]:=16#5a23;
    unicode[1256]:=16#5a25;
    unicode[1257]:=16#5a29;
    unicode[1258]:=16#5a31;
    unicode[1259]:=16#5a32;
    unicode[1260]:=16#5a34;
    unicode[1261]:=16#5a36;
    unicode[1262]:=16#5a3c;
    unicode[1263]:=16#5a40;
    unicode[1264]:=16#5a46;
    unicode[1265]:=16#5a49;
    unicode[1266]:=16#5a4a;
    unicode[1267]:=16#5a55;
    unicode[1268]:=16#5a5a;
    unicode[1269]:=16#5a62;
    unicode[1270]:=16#5a67;
    unicode[1271]:=16#5a6a;
    unicode[1272]:=16#5a74;
    unicode[1273]:=16#5a75;
    unicode[1274]:=16#5a76;
    unicode[1275]:=16#5a77;
    unicode[1276]:=16#5a7a;
    unicode[1277]:=16#5a7f;
    unicode[1278]:=16#5a92;
    unicode[1279]:=16#5a9a;
    unicode[1280]:=16#5a9b;
    unicode[1281]:=16#5aaa;
    unicode[1282]:=16#5ab2;
    unicode[1283]:=16#5ab3;
    unicode[1284]:=16#5ab5;
    unicode[1285]:=16#5ab8;
    unicode[1286]:=16#5abe;
    unicode[1287]:=16#5ac1;
    unicode[1288]:=16#5ac2;
    unicode[1289]:=16#5ac9;
    unicode[1290]:=16#5acc;
    unicode[1291]:=16#5ad2;
    unicode[1292]:=16#5ad4;
    unicode[1293]:=16#5ad6;
    unicode[1294]:=16#5ad8;
    unicode[1295]:=16#5adc;
    unicode[1296]:=16#5ae0;
    unicode[1297]:=16#5ae1;
    unicode[1298]:=16#5ae3;
    unicode[1299]:=16#5ae6;
    unicode[1300]:=16#5ae9;
    unicode[1301]:=16#5aeb;
    unicode[1302]:=16#5af1;
    unicode[1303]:=16#5b09;
    unicode[1304]:=16#5b16;
    unicode[1305]:=16#5b17;
    unicode[1306]:=16#5b32;
    unicode[1307]:=16#5b34;
    unicode[1308]:=16#5b37;
    unicode[1309]:=16#5b40;
    unicode[1310]:=16#5b50;
    unicode[1311]:=16#5b51;
    unicode[1312]:=16#5b53;
    unicode[1313]:=16#5b54;
    unicode[1314]:=16#5b55;
    unicode[1315]:=16#5b57;
    unicode[1316]:=16#5b58;
    unicode[1317]:=16#5b59;
    unicode[1318]:=16#5b5a;
    unicode[1319]:=16#5b5b;
    unicode[1320]:=16#5b5c;
    unicode[1321]:=16#5b5d;
    unicode[1322]:=16#5b5f;
    unicode[1323]:=16#5b62;
    unicode[1324]:=16#5b63;
    unicode[1325]:=16#5b64;
    unicode[1326]:=16#5b65;
    unicode[1327]:=16#5b66;
    unicode[1328]:=16#5b69;
    unicode[1329]:=16#5b6a;
    unicode[1330]:=16#5b6c;
    unicode[1331]:=16#5b70;
    unicode[1332]:=16#5b71;
    unicode[1333]:=16#5b73;
    unicode[1334]:=16#5b75;
    unicode[1335]:=16#5b7a;
    unicode[1336]:=16#5b7d;
    unicode[1337]:=16#5b80;
    unicode[1338]:=16#5b81;
    unicode[1339]:=16#5b83;
    unicode[1340]:=16#5b84;
    unicode[1341]:=16#5b85;
    unicode[1342]:=16#5b87;
    unicode[1343]:=16#5b88;
    unicode[1344]:=16#5b89;
    unicode[1345]:=16#5b8b;
    unicode[1346]:=16#5b8c;
    unicode[1347]:=16#5b8f;
    unicode[1348]:=16#5b93;
    unicode[1349]:=16#5b95;
    unicode[1350]:=16#5b97;
    unicode[1351]:=16#5b98;
    unicode[1352]:=16#5b99;
    unicode[1353]:=16#5b9a;
    unicode[1354]:=16#5b9b;
    unicode[1355]:=16#5b9c;
    unicode[1356]:=16#5b9d;
    unicode[1357]:=16#5b9e;
    unicode[1358]:=16#5ba0;
    unicode[1359]:=16#5ba1;
    unicode[1360]:=16#5ba2;
    unicode[1361]:=16#5ba3;
    unicode[1362]:=16#5ba4;
    unicode[1363]:=16#5ba5;
    unicode[1364]:=16#5ba6;
    unicode[1365]:=16#5baa;
    unicode[1366]:=16#5bab;
    unicode[1367]:=16#5bb0;
    unicode[1368]:=16#5bb3;
    unicode[1369]:=16#5bb4;
    unicode[1370]:=16#5bb5;
    unicode[1371]:=16#5bb6;
    unicode[1372]:=16#5bb8;
    unicode[1373]:=16#5bb9;
    unicode[1374]:=16#5bbd;
    unicode[1375]:=16#5bbe;
    unicode[1376]:=16#5bbf;
    unicode[1377]:=16#5bc2;
    unicode[1378]:=16#5bc4;
    unicode[1379]:=16#5bc5;
    unicode[1380]:=16#5bc6;
    unicode[1381]:=16#5bc7;
    unicode[1382]:=16#5bcc;
    unicode[1383]:=16#5bd0;
    unicode[1384]:=16#5bd2;
    unicode[1385]:=16#5bd3;
    unicode[1386]:=16#5bdd;
    unicode[1387]:=16#5bde;
    unicode[1388]:=16#5bdf;
    unicode[1389]:=16#5be1;
    unicode[1390]:=16#5be4;
    unicode[1391]:=16#5be5;
    unicode[1392]:=16#5be8;
    unicode[1393]:=16#5bee;
    unicode[1394]:=16#5bf0;
    unicode[1395]:=16#5bf8;
    unicode[1396]:=16#5bf9;
    unicode[1397]:=16#5bfa;
    unicode[1398]:=16#5bfb;
    unicode[1399]:=16#5bfc;
    unicode[1400]:=16#5bff;
    unicode[1401]:=16#5c01;
    unicode[1402]:=16#5c04;
    unicode[1403]:=16#5c06;
    unicode[1404]:=16#5c09;
    unicode[1405]:=16#5c0a;
    unicode[1406]:=16#5c0f;
    unicode[1407]:=16#5c11;
    unicode[1408]:=16#5c14;
    unicode[1409]:=16#5c15;
    unicode[1410]:=16#5c16;
    unicode[1411]:=16#5c18;
    unicode[1412]:=16#5c1a;
    unicode[1413]:=16#5c1c;
    unicode[1414]:=16#5c1d;
    unicode[1415]:=16#5c22;
    unicode[1416]:=16#5c24;
    unicode[1417]:=16#5c25;
    unicode[1418]:=16#5c27;
    unicode[1419]:=16#5c2c;
    unicode[1420]:=16#5c31;
    unicode[1421]:=16#5c34;
    unicode[1422]:=16#5c38;
    unicode[1423]:=16#5c39;
    unicode[1424]:=16#5c3a;
    unicode[1425]:=16#5c3b;
    unicode[1426]:=16#5c3c;
    unicode[1427]:=16#5c3d;
    unicode[1428]:=16#5c3e;
    unicode[1429]:=16#5c3f;
    unicode[1430]:=16#5c40;
    unicode[1431]:=16#5c41;
    unicode[1432]:=16#5c42;
    unicode[1433]:=16#5c45;
    unicode[1434]:=16#5c48;
    unicode[1435]:=16#5c49;
    unicode[1436]:=16#5c4a;
    unicode[1437]:=16#5c4b;
    unicode[1438]:=16#5c4e;
    unicode[1439]:=16#5c4f;
    unicode[1440]:=16#5c50;
    unicode[1441]:=16#5c51;
    unicode[1442]:=16#5c55;
    unicode[1443]:=16#5c59;
    unicode[1444]:=16#5c5e;
    unicode[1445]:=16#5c60;
    unicode[1446]:=16#5c61;
    unicode[1447]:=16#5c63;
    unicode[1448]:=16#5c65;
    unicode[1449]:=16#5c66;
    unicode[1450]:=16#5c6e;
    unicode[1451]:=16#5c6f;
    unicode[1452]:=16#5c71;
    unicode[1453]:=16#5c79;
    unicode[1454]:=16#5c7a;
    unicode[1455]:=16#5c7f;
    unicode[1456]:=16#5c81;
    unicode[1457]:=16#5c82;
    unicode[1458]:=16#5c88;
    unicode[1459]:=16#5c8c;
    unicode[1460]:=16#5c8d;
    unicode[1461]:=16#5c90;
    unicode[1462]:=16#5c91;
    unicode[1463]:=16#5c94;
    unicode[1464]:=16#5c96;
    unicode[1465]:=16#5c97;
    unicode[1466]:=16#5c98;
    unicode[1467]:=16#5c99;
    unicode[1468]:=16#5c9a;
    unicode[1469]:=16#5c9b;
    unicode[1470]:=16#5c9c;
    unicode[1471]:=16#5ca2;
    unicode[1472]:=16#5ca3;
    unicode[1473]:=16#5ca9;
    unicode[1474]:=16#5cab;
    unicode[1475]:=16#5cac;
    unicode[1476]:=16#5cad;
    unicode[1477]:=16#5cb1;
    unicode[1478]:=16#5cb3;
    unicode[1479]:=16#5cb5;
    unicode[1480]:=16#5cb7;
    unicode[1481]:=16#5cb8;
    unicode[1482]:=16#5cbd;
    unicode[1483]:=16#5cbf;
    unicode[1484]:=16#5cc1;
    unicode[1485]:=16#5cc4;
    unicode[1486]:=16#5ccb;
    unicode[1487]:=16#5cd2;
    unicode[1488]:=16#5cd9;
    unicode[1489]:=16#5ce1;
    unicode[1490]:=16#5ce4;
    unicode[1491]:=16#5ce5;
    unicode[1492]:=16#5ce6;
    unicode[1493]:=16#5ce8;
    unicode[1494]:=16#5cea;
    unicode[1495]:=16#5ced;
    unicode[1496]:=16#5cf0;
    unicode[1497]:=16#5cfb;
    unicode[1498]:=16#5d02;
    unicode[1499]:=16#5d03;
    unicode[1500]:=16#5d06;
    unicode[1501]:=16#5d07;
    unicode[1502]:=16#5d0e;
    unicode[1503]:=16#5d14;
    unicode[1504]:=16#5d16;
    unicode[1505]:=16#5d1b;
    unicode[1506]:=16#5d1e;
    unicode[1507]:=16#5d24;
    unicode[1508]:=16#5d26;
    unicode[1509]:=16#5d27;
    unicode[1510]:=16#5d29;
    unicode[1511]:=16#5d2d;
    unicode[1512]:=16#5d2e;
    unicode[1513]:=16#5d34;
    unicode[1514]:=16#5d3d;
    unicode[1515]:=16#5d3e;
    unicode[1516]:=16#5d47;
    unicode[1517]:=16#5d4a;
    unicode[1518]:=16#5d4b;
    unicode[1519]:=16#5d4c;
    unicode[1520]:=16#5d58;
    unicode[1521]:=16#5d5b;
    unicode[1522]:=16#5d5d;
    unicode[1523]:=16#5d69;
    unicode[1524]:=16#5d6b;
    unicode[1525]:=16#5d6c;
    unicode[1526]:=16#5d6f;
    unicode[1527]:=16#5d74;
    unicode[1528]:=16#5d82;
    unicode[1529]:=16#5d99;
    unicode[1530]:=16#5d9d;
    unicode[1531]:=16#5db7;
    unicode[1532]:=16#5dc5;
    unicode[1533]:=16#5dcd;
    unicode[1534]:=16#5ddb;
    unicode[1535]:=16#5ddd;
    unicode[1536]:=16#5dde;
    unicode[1537]:=16#5de1;
    unicode[1538]:=16#5de2;
    unicode[1539]:=16#5de5;
    unicode[1540]:=16#5de6;
    unicode[1541]:=16#5de7;
    unicode[1542]:=16#5de8;
    unicode[1543]:=16#5de9;
    unicode[1544]:=16#5deb;
    unicode[1545]:=16#5dee;
    unicode[1546]:=16#5def;
    unicode[1547]:=16#5df1;
    unicode[1548]:=16#5df2;
    unicode[1549]:=16#5df3;
    unicode[1550]:=16#5df4;
    unicode[1551]:=16#5df7;
    unicode[1552]:=16#5dfd;
    unicode[1553]:=16#5dfe;
    unicode[1554]:=16#5e01;
    unicode[1555]:=16#5e02;
    unicode[1556]:=16#5e03;
    unicode[1557]:=16#5e05;
    unicode[1558]:=16#5e06;
    unicode[1559]:=16#5e08;
    unicode[1560]:=16#5e0c;
    unicode[1561]:=16#5e0f;
    unicode[1562]:=16#5e10;
    unicode[1563]:=16#5e11;
    unicode[1564]:=16#5e14;
    unicode[1565]:=16#5e15;
    unicode[1566]:=16#5e16;
    unicode[1567]:=16#5e18;
    unicode[1568]:=16#5e19;
    unicode[1569]:=16#5e1a;
    unicode[1570]:=16#5e1b;
    unicode[1571]:=16#5e1c;
    unicode[1572]:=16#5e1d;
    unicode[1573]:=16#5e26;
    unicode[1574]:=16#5e27;
    unicode[1575]:=16#5e2d;
    unicode[1576]:=16#5e2e;
    unicode[1577]:=16#5e31;
    unicode[1578]:=16#5e37;
    unicode[1579]:=16#5e38;
    unicode[1580]:=16#5e3b;
    unicode[1581]:=16#5e3c;
    unicode[1582]:=16#5e3d;
    unicode[1583]:=16#5e42;
    unicode[1584]:=16#5e44;
    unicode[1585]:=16#5e45;
    unicode[1586]:=16#5e4c;
    unicode[1587]:=16#5e54;
    unicode[1588]:=16#5e55;
    unicode[1589]:=16#5e5b;
    unicode[1590]:=16#5e5e;
    unicode[1591]:=16#5e61;
    unicode[1592]:=16#5e62;
    unicode[1593]:=16#5e72;
    unicode[1594]:=16#5e73;
    unicode[1595]:=16#5e74;
    unicode[1596]:=16#5e76;
    unicode[1597]:=16#5e78;
    unicode[1598]:=16#5e7a;
    unicode[1599]:=16#5e7b;
    unicode[1600]:=16#5e7c;
    unicode[1601]:=16#5e7d;
    unicode[1602]:=16#5e7f;
    unicode[1603]:=16#5e80;
    unicode[1604]:=16#5e84;
    unicode[1605]:=16#5e86;
    unicode[1606]:=16#5e87;
    unicode[1607]:=16#5e8a;
    unicode[1608]:=16#5e8b;
    unicode[1609]:=16#5e8f;
    unicode[1610]:=16#5e90;
    unicode[1611]:=16#5e91;
    unicode[1612]:=16#5e93;
    unicode[1613]:=16#5e94;
    unicode[1614]:=16#5e95;
    unicode[1615]:=16#5e96;
    unicode[1616]:=16#5e97;
    unicode[1617]:=16#5e99;
    unicode[1618]:=16#5e9a;
    unicode[1619]:=16#5e9c;
    unicode[1620]:=16#5e9e;
    unicode[1621]:=16#5e9f;
    unicode[1622]:=16#5ea0;
    unicode[1623]:=16#5ea5;
    unicode[1624]:=16#5ea6;
    unicode[1625]:=16#5ea7;
    unicode[1626]:=16#5ead;
    unicode[1627]:=16#5eb3;
    unicode[1628]:=16#5eb5;
    unicode[1629]:=16#5eb6;
    unicode[1630]:=16#5eb7;
    unicode[1631]:=16#5eb8;
    unicode[1632]:=16#5eb9;
    unicode[1633]:=16#5ebe;
    unicode[1634]:=16#5ec9;
    unicode[1635]:=16#5eca;
    unicode[1636]:=16#5ed1;
    unicode[1637]:=16#5ed2;
    unicode[1638]:=16#5ed3;
    unicode[1639]:=16#5ed6;
    unicode[1640]:=16#5edb;
    unicode[1641]:=16#5ee8;
    unicode[1642]:=16#5eea;
    unicode[1643]:=16#5ef4;
    unicode[1644]:=16#5ef6;
    unicode[1645]:=16#5ef7;
    unicode[1646]:=16#5efa;
    unicode[1647]:=16#5efe;
    unicode[1648]:=16#5eff;
    unicode[1649]:=16#5f00;
    unicode[1650]:=16#5f01;
    unicode[1651]:=16#5f02;
    unicode[1652]:=16#5f03;
    unicode[1653]:=16#5f04;
    unicode[1654]:=16#5f08;
    unicode[1655]:=16#5f0a;
    unicode[1656]:=16#5f0b;
    unicode[1657]:=16#5f0f;
    unicode[1658]:=16#5f11;
    unicode[1659]:=16#5f13;
    unicode[1660]:=16#5f15;
    unicode[1661]:=16#5f17;
    unicode[1662]:=16#5f18;
    unicode[1663]:=16#5f1b;
    unicode[1664]:=16#5f1f;
    unicode[1665]:=16#5f20;
    unicode[1666]:=16#5f25;
    unicode[1667]:=16#5f26;
    unicode[1668]:=16#5f27;
    unicode[1669]:=16#5f29;
    unicode[1670]:=16#5f2a;
    unicode[1671]:=16#5f2d;
    unicode[1672]:=16#5f2f;
    unicode[1673]:=16#5f31;
    unicode[1674]:=16#5f39;
    unicode[1675]:=16#5f3a;
    unicode[1676]:=16#5f3c;
    unicode[1677]:=16#5f40;
    unicode[1678]:=16#5f50;
    unicode[1679]:=16#5f52;
    unicode[1680]:=16#5f53;
    unicode[1681]:=16#5f55;
    unicode[1682]:=16#5f56;
    unicode[1683]:=16#5f57;
    unicode[1684]:=16#5f58;
    unicode[1685]:=16#5f5d;
    unicode[1686]:=16#5f61;
    unicode[1687]:=16#5f62;
    unicode[1688]:=16#5f64;
    unicode[1689]:=16#5f66;
    unicode[1690]:=16#5f69;
    unicode[1691]:=16#5f6a;
    unicode[1692]:=16#5f6c;
    unicode[1693]:=16#5f6d;
    unicode[1694]:=16#5f70;
    unicode[1695]:=16#5f71;
    unicode[1696]:=16#5f73;
    unicode[1697]:=16#5f77;
    unicode[1698]:=16#5f79;
    unicode[1699]:=16#5f7b;
    unicode[1700]:=16#5f7c;
    unicode[1701]:=16#5f80;
    unicode[1702]:=16#5f81;
    unicode[1703]:=16#5f82;
    unicode[1704]:=16#5f84;
    unicode[1705]:=16#5f85;
    unicode[1706]:=16#5f87;
    unicode[1707]:=16#5f88;
    unicode[1708]:=16#5f89;
    unicode[1709]:=16#5f8a;
    unicode[1710]:=16#5f8b;
    unicode[1711]:=16#5f8c;
    unicode[1712]:=16#5f90;
    unicode[1713]:=16#5f92;
    unicode[1714]:=16#5f95;
    unicode[1715]:=16#5f97;
    unicode[1716]:=16#5f98;
    unicode[1717]:=16#5f99;
    unicode[1718]:=16#5f9c;
    unicode[1719]:=16#5fa1;
    unicode[1720]:=16#5fa8;
    unicode[1721]:=16#5faa;
    unicode[1722]:=16#5fad;
    unicode[1723]:=16#5fae;
    unicode[1724]:=16#5fb5;
    unicode[1725]:=16#5fb7;
    unicode[1726]:=16#5fbc;
    unicode[1727]:=16#5fbd;
    unicode[1728]:=16#5fc3;
    unicode[1729]:=16#5fc4;
    unicode[1730]:=16#5fc5;
    unicode[1731]:=16#5fc6;
    unicode[1732]:=16#5fc9;
    unicode[1733]:=16#5fcc;
    unicode[1734]:=16#5fcd;
    unicode[1735]:=16#5fcf;
    unicode[1736]:=16#5fd0;
    unicode[1737]:=16#5fd1;
    unicode[1738]:=16#5fd2;
    unicode[1739]:=16#5fd6;
    unicode[1740]:=16#5fd7;
    unicode[1741]:=16#5fd8;
    unicode[1742]:=16#5fd9;
    unicode[1743]:=16#5fdd;
    unicode[1744]:=16#5fe0;
    unicode[1745]:=16#5fe1;
    unicode[1746]:=16#5fe4;
    unicode[1747]:=16#5fe7;
    unicode[1748]:=16#5fea;
    unicode[1749]:=16#5feb;
    unicode[1750]:=16#5fed;
    unicode[1751]:=16#5fee;
    unicode[1752]:=16#5ff1;
    unicode[1753]:=16#5ff5;
    unicode[1754]:=16#5ff8;
    unicode[1755]:=16#5ffb;
    unicode[1756]:=16#5ffd;
    unicode[1757]:=16#5ffe;
    unicode[1758]:=16#5fff;
    unicode[1759]:=16#6000;
    unicode[1760]:=16#6001;
    unicode[1761]:=16#6002;
    unicode[1762]:=16#6003;
    unicode[1763]:=16#6004;
    unicode[1764]:=16#6005;
    unicode[1765]:=16#6006;
    unicode[1766]:=16#600a;
    unicode[1767]:=16#600d;
    unicode[1768]:=16#600e;
    unicode[1769]:=16#600f;
    unicode[1770]:=16#6012;
    unicode[1771]:=16#6014;
    unicode[1772]:=16#6015;
    unicode[1773]:=16#6016;
    unicode[1774]:=16#6019;
    unicode[1775]:=16#601b;
    unicode[1776]:=16#601c;
    unicode[1777]:=16#601d;
    unicode[1778]:=16#6020;
    unicode[1779]:=16#6021;
    unicode[1780]:=16#6025;
    unicode[1781]:=16#6026;
    unicode[1782]:=16#6027;
    unicode[1783]:=16#6028;
    unicode[1784]:=16#6029;
    unicode[1785]:=16#602a;
    unicode[1786]:=16#602b;
    unicode[1787]:=16#602f;
    unicode[1788]:=16#6035;
    unicode[1789]:=16#603b;
    unicode[1790]:=16#603c;
    unicode[1791]:=16#603f;
    unicode[1792]:=16#6041;
    unicode[1793]:=16#6042;
    unicode[1794]:=16#6043;
    unicode[1795]:=16#604b;
    unicode[1796]:=16#604d;
    unicode[1797]:=16#6050;
    unicode[1798]:=16#6052;
    unicode[1799]:=16#6055;
    unicode[1800]:=16#6059;
    unicode[1801]:=16#605a;
    unicode[1802]:=16#605d;
    unicode[1803]:=16#6062;
    unicode[1804]:=16#6063;
    unicode[1805]:=16#6064;
    unicode[1806]:=16#6067;
    unicode[1807]:=16#6068;
    unicode[1808]:=16#6069;
    unicode[1809]:=16#606a;
    unicode[1810]:=16#606b;
    unicode[1811]:=16#606c;
    unicode[1812]:=16#606d;
    unicode[1813]:=16#606f;
    unicode[1814]:=16#6070;
    unicode[1815]:=16#6073;
    unicode[1816]:=16#6076;
    unicode[1817]:=16#6078;
    unicode[1818]:=16#6079;
    unicode[1819]:=16#607a;
    unicode[1820]:=16#607b;
    unicode[1821]:=16#607c;
    unicode[1822]:=16#607d;
    unicode[1823]:=16#607f;
    unicode[1824]:=16#6083;
    unicode[1825]:=16#6084;
    unicode[1826]:=16#6089;
    unicode[1827]:=16#608c;
    unicode[1828]:=16#608d;
    unicode[1829]:=16#6092;
    unicode[1830]:=16#6094;
    unicode[1831]:=16#6096;
    unicode[1832]:=16#609a;
    unicode[1833]:=16#609b;
    unicode[1834]:=16#609d;
    unicode[1835]:=16#609f;
    unicode[1836]:=16#60a0;
    unicode[1837]:=16#60a3;
    unicode[1838]:=16#60a6;
    unicode[1839]:=16#60a8;
    unicode[1840]:=16#60ab;
    unicode[1841]:=16#60ac;
    unicode[1842]:=16#60ad;
    unicode[1843]:=16#60af;
    unicode[1844]:=16#60b1;
    unicode[1845]:=16#60b2;
    unicode[1846]:=16#60b4;
    unicode[1847]:=16#60b8;
    unicode[1848]:=16#60bb;
    unicode[1849]:=16#60bc;
    unicode[1850]:=16#60c5;
    unicode[1851]:=16#60c6;
    unicode[1852]:=16#60ca;
    unicode[1853]:=16#60cb;
    unicode[1854]:=16#60d1;
    unicode[1855]:=16#60d5;
    unicode[1856]:=16#60d8;
    unicode[1857]:=16#60da;
    unicode[1858]:=16#60dc;
    unicode[1859]:=16#60dd;
    unicode[1860]:=16#60df;
    unicode[1861]:=16#60e0;
    unicode[1862]:=16#60e6;
    unicode[1863]:=16#60e7;
    unicode[1864]:=16#60e8;
    unicode[1865]:=16#60e9;
    unicode[1866]:=16#60eb;
    unicode[1867]:=16#60ec;
    unicode[1868]:=16#60ed;
    unicode[1869]:=16#60ee;
    unicode[1870]:=16#60ef;
    unicode[1871]:=16#60f0;
    unicode[1872]:=16#60f3;
    unicode[1873]:=16#60f4;
    unicode[1874]:=16#60f6;
    unicode[1875]:=16#60f9;
    unicode[1876]:=16#60fa;
    unicode[1877]:=16#6100;
    unicode[1878]:=16#6101;
    unicode[1879]:=16#6106;
    unicode[1880]:=16#6108;
    unicode[1881]:=16#6109;
    unicode[1882]:=16#610d;
    unicode[1883]:=16#610e;
    unicode[1884]:=16#610f;
    unicode[1885]:=16#6115;
    unicode[1886]:=16#611a;
    unicode[1887]:=16#611f;
    unicode[1888]:=16#6120;
    unicode[1889]:=16#6123;
    unicode[1890]:=16#6124;
    unicode[1891]:=16#6126;
    unicode[1892]:=16#6127;
    unicode[1893]:=16#612b;
    unicode[1894]:=16#613f;
    unicode[1895]:=16#6148;
    unicode[1896]:=16#614a;
    unicode[1897]:=16#614c;
    unicode[1898]:=16#614e;
    unicode[1899]:=16#6151;
    unicode[1900]:=16#6155;
    unicode[1901]:=16#615d;
    unicode[1902]:=16#6162;
    unicode[1903]:=16#6167;
    unicode[1904]:=16#6168;
    unicode[1905]:=16#6170;
    unicode[1906]:=16#6175;
    unicode[1907]:=16#6177;
    unicode[1908]:=16#618b;
    unicode[1909]:=16#618e;
    unicode[1910]:=16#6194;
    unicode[1911]:=16#619d;
    unicode[1912]:=16#61a7;
    unicode[1913]:=16#61a8;
    unicode[1914]:=16#61a9;
    unicode[1915]:=16#61ac;
    unicode[1916]:=16#61b7;
    unicode[1917]:=16#61be;
    unicode[1918]:=16#61c2;
    unicode[1919]:=16#61c8;
    unicode[1920]:=16#61ca;
    unicode[1921]:=16#61cb;
    unicode[1922]:=16#61d1;
    unicode[1923]:=16#61d2;
    unicode[1924]:=16#61d4;
    unicode[1925]:=16#61e6;
    unicode[1926]:=16#61f5;
    unicode[1927]:=16#61ff;
    unicode[1928]:=16#6206;
    unicode[1929]:=16#6208;
    unicode[1930]:=16#620a;
    unicode[1931]:=16#620b;
    unicode[1932]:=16#620c;
    unicode[1933]:=16#620d;
    unicode[1934]:=16#620e;
    unicode[1935]:=16#620f;
    unicode[1936]:=16#6210;
    unicode[1937]:=16#6211;
    unicode[1938]:=16#6212;
    unicode[1939]:=16#6215;
    unicode[1940]:=16#6216;
    unicode[1941]:=16#6217;
    unicode[1942]:=16#6218;
    unicode[1943]:=16#621a;
    unicode[1944]:=16#621b;
    unicode[1945]:=16#621f;
    unicode[1946]:=16#6221;
    unicode[1947]:=16#6222;
    unicode[1948]:=16#6224;
    unicode[1949]:=16#6225;
    unicode[1950]:=16#622a;
    unicode[1951]:=16#622c;
    unicode[1952]:=16#622e;
    unicode[1953]:=16#6233;
    unicode[1954]:=16#6234;
    unicode[1955]:=16#6237;
    unicode[1956]:=16#623d;
    unicode[1957]:=16#623e;
    unicode[1958]:=16#623f;
    unicode[1959]:=16#6240;
    unicode[1960]:=16#6241;
    unicode[1961]:=16#6243;
    unicode[1962]:=16#6247;
    unicode[1963]:=16#6248;
    unicode[1964]:=16#6249;
    unicode[1965]:=16#624b;
    unicode[1966]:=16#624c;
    unicode[1967]:=16#624d;
    unicode[1968]:=16#624e;
    unicode[1969]:=16#6251;
    unicode[1970]:=16#6252;
    unicode[1971]:=16#6253;
    unicode[1972]:=16#6254;
    unicode[1973]:=16#6258;
    unicode[1974]:=16#625b;
    unicode[1975]:=16#6263;
    unicode[1976]:=16#6266;
    unicode[1977]:=16#6267;
    unicode[1978]:=16#6269;
    unicode[1979]:=16#626a;
    unicode[1980]:=16#626b;
    unicode[1981]:=16#626c;
    unicode[1982]:=16#626d;
    unicode[1983]:=16#626e;
    unicode[1984]:=16#626f;
    unicode[1985]:=16#6270;
    unicode[1986]:=16#6273;
    unicode[1987]:=16#6276;
    unicode[1988]:=16#6279;
    unicode[1989]:=16#627c;
    unicode[1990]:=16#627e;
    unicode[1991]:=16#627f;
    unicode[1992]:=16#6280;
    unicode[1993]:=16#6284;
    unicode[1994]:=16#6289;
    unicode[1995]:=16#628a;
    unicode[1996]:=16#6291;
    unicode[1997]:=16#6292;
    unicode[1998]:=16#6293;
    unicode[1999]:=16#6295;        //unicode码 1000-1999
END_IF;
(* Rung 6 *)
IF P_On THEN
    unicode[2000]:=16#6296;
    unicode[2001]:=16#6297;
    unicode[2002]:=16#6298;
    unicode[2003]:=16#629a;
    unicode[2004]:=16#629b;
    unicode[2005]:=16#629f;
    unicode[2006]:=16#62a0;
    unicode[2007]:=16#62a1;
    unicode[2008]:=16#62a2;
    unicode[2009]:=16#62a4;
    unicode[2010]:=16#62a5;
    unicode[2011]:=16#62a8;
    unicode[2012]:=16#62ab;
    unicode[2013]:=16#62ac;
    unicode[2014]:=16#62b1;
    unicode[2015]:=16#62b5;
    unicode[2016]:=16#62b9;
    unicode[2017]:=16#62bb;
    unicode[2018]:=16#62bc;
    unicode[2019]:=16#62bd;
    unicode[2020]:=16#62bf;
    unicode[2021]:=16#62c2;
    unicode[2022]:=16#62c4;
    unicode[2023]:=16#62c5;
    unicode[2024]:=16#62c6;
    unicode[2025]:=16#62c7;
    unicode[2026]:=16#62c8;
    unicode[2027]:=16#62c9;
    unicode[2028]:=16#62ca;
    unicode[2029]:=16#62cc;
    unicode[2030]:=16#62cd;
    unicode[2031]:=16#62ce;
    unicode[2032]:=16#62d0;
    unicode[2033]:=16#62d2;
    unicode[2034]:=16#62d3;
    unicode[2035]:=16#62d4;
    unicode[2036]:=16#62d6;
    unicode[2037]:=16#62d7;
    unicode[2038]:=16#62d8;
    unicode[2039]:=16#62d9;
    unicode[2040]:=16#62da;
    unicode[2041]:=16#62db;
    unicode[2042]:=16#62dc;
    unicode[2043]:=16#62df;
    unicode[2044]:=16#62e2;
    unicode[2045]:=16#62e3;
    unicode[2046]:=16#62e5;
    unicode[2047]:=16#62e6;
    unicode[2048]:=16#62e7;
    unicode[2049]:=16#62e8;
    unicode[2050]:=16#62e9;
    unicode[2051]:=16#62ec;
    unicode[2052]:=16#62ed;
    unicode[2053]:=16#62ee;
    unicode[2054]:=16#62ef;
    unicode[2055]:=16#62f1;
    unicode[2056]:=16#62f3;
    unicode[2057]:=16#62f4;
    unicode[2058]:=16#62f6;
    unicode[2059]:=16#62f7;
    unicode[2060]:=16#62fc;
    unicode[2061]:=16#62fd;
    unicode[2062]:=16#62fe;
    unicode[2063]:=16#62ff;
    unicode[2064]:=16#6301;
    unicode[2065]:=16#6302;
    unicode[2066]:=16#6307;
    unicode[2067]:=16#6308;
    unicode[2068]:=16#6309;
    unicode[2069]:=16#630e;
    unicode[2070]:=16#6311;
    unicode[2071]:=16#6316;
    unicode[2072]:=16#631a;
    unicode[2073]:=16#631b;
    unicode[2074]:=16#631d;
    unicode[2075]:=16#631e;
    unicode[2076]:=16#631f;
    unicode[2077]:=16#6320;
    unicode[2078]:=16#6321;
    unicode[2079]:=16#6322;
    unicode[2080]:=16#6323;
    unicode[2081]:=16#6324;
    unicode[2082]:=16#6325;
    unicode[2083]:=16#6328;
    unicode[2084]:=16#632a;
    unicode[2085]:=16#632b;
    unicode[2086]:=16#632f;
    unicode[2087]:=16#6332;
    unicode[2088]:=16#6339;
    unicode[2089]:=16#633a;
    unicode[2090]:=16#633d;
    unicode[2091]:=16#6342;
    unicode[2092]:=16#6343;
    unicode[2093]:=16#6345;
    unicode[2094]:=16#6346;
    unicode[2095]:=16#6349;
    unicode[2096]:=16#634b;
    unicode[2097]:=16#634c;
    unicode[2098]:=16#634d;
    unicode[2099]:=16#634e;
    unicode[2100]:=16#634f;
    unicode[2101]:=16#6350;
    unicode[2102]:=16#6355;
    unicode[2103]:=16#635e;
    unicode[2104]:=16#635f;
    unicode[2105]:=16#6361;
    unicode[2106]:=16#6362;
    unicode[2107]:=16#6363;
    unicode[2108]:=16#6367;
    unicode[2109]:=16#6369;
    unicode[2110]:=16#636d;
    unicode[2111]:=16#636e;
    unicode[2112]:=16#6371;
    unicode[2113]:=16#6376;
    unicode[2114]:=16#6377;
    unicode[2115]:=16#637a;
    unicode[2116]:=16#637b;
    unicode[2117]:=16#6380;
    unicode[2118]:=16#6382;
    unicode[2119]:=16#6387;
    unicode[2120]:=16#6388;
    unicode[2121]:=16#6389;
    unicode[2122]:=16#638a;
    unicode[2123]:=16#638c;
    unicode[2124]:=16#638e;
    unicode[2125]:=16#638f;
    unicode[2126]:=16#6390;
    unicode[2127]:=16#6392;
    unicode[2128]:=16#6396;
    unicode[2129]:=16#6398;
    unicode[2130]:=16#63a0;
    unicode[2131]:=16#63a2;
    unicode[2132]:=16#63a3;
    unicode[2133]:=16#63a5;
    unicode[2134]:=16#63a7;
    unicode[2135]:=16#63a8;
    unicode[2136]:=16#63a9;
    unicode[2137]:=16#63aa;
    unicode[2138]:=16#63ac;
    unicode[2139]:=16#63ad;
    unicode[2140]:=16#63ae;
    unicode[2141]:=16#63b0;
    unicode[2142]:=16#63b3;
    unicode[2143]:=16#63b4;
    unicode[2144]:=16#63b7;
    unicode[2145]:=16#63b8;
    unicode[2146]:=16#63ba;
    unicode[2147]:=16#63bc;
    unicode[2148]:=16#63be;
    unicode[2149]:=16#63c4;
    unicode[2150]:=16#63c6;
    unicode[2151]:=16#63c9;
    unicode[2152]:=16#63cd;
    unicode[2153]:=16#63ce;
    unicode[2154]:=16#63cf;
    unicode[2155]:=16#63d0;
    unicode[2156]:=16#63d2;
    unicode[2157]:=16#63d6;
    unicode[2158]:=16#63de;
    unicode[2159]:=16#63e0;
    unicode[2160]:=16#63e1;
    unicode[2161]:=16#63e3;
    unicode[2162]:=16#63e9;
    unicode[2163]:=16#63ea;
    unicode[2164]:=16#63ed;
    unicode[2165]:=16#63f2;
    unicode[2166]:=16#63f4;
    unicode[2167]:=16#63f6;
    unicode[2168]:=16#63f8;
    unicode[2169]:=16#63fd;
    unicode[2170]:=16#63ff;
    unicode[2171]:=16#6400;
    unicode[2172]:=16#6401;
    unicode[2173]:=16#6402;
    unicode[2174]:=16#6405;
    unicode[2175]:=16#640b;
    unicode[2176]:=16#640c;
    unicode[2177]:=16#640f;
    unicode[2178]:=16#6410;
    unicode[2179]:=16#6413;
    unicode[2180]:=16#6414;
    unicode[2181]:=16#641b;
    unicode[2182]:=16#641c;
    unicode[2183]:=16#641e;
    unicode[2184]:=16#6420;
    unicode[2185]:=16#6421;
    unicode[2186]:=16#6426;
    unicode[2187]:=16#642a;
    unicode[2188]:=16#642c;
    unicode[2189]:=16#642d;
    unicode[2190]:=16#6434;
    unicode[2191]:=16#643a;
    unicode[2192]:=16#643d;
    unicode[2193]:=16#643f;
    unicode[2194]:=16#6441;
    unicode[2195]:=16#6444;
    unicode[2196]:=16#6445;
    unicode[2197]:=16#6446;
    unicode[2198]:=16#6447;
    unicode[2199]:=16#6448;
    unicode[2200]:=16#644a;
    unicode[2201]:=16#6452;
    unicode[2202]:=16#6454;
    unicode[2203]:=16#6458;
    unicode[2204]:=16#645e;
    unicode[2205]:=16#6467;
    unicode[2206]:=16#6469;
    unicode[2207]:=16#646d;
    unicode[2208]:=16#6478;
    unicode[2209]:=16#6479;
    unicode[2210]:=16#647a;
    unicode[2211]:=16#6482;
    unicode[2212]:=16#6484;
    unicode[2213]:=16#6485;
    unicode[2214]:=16#6487;
    unicode[2215]:=16#6491;
    unicode[2216]:=16#6492;
    unicode[2217]:=16#6495;
    unicode[2218]:=16#6496;
    unicode[2219]:=16#6499;
    unicode[2220]:=16#649e;
    unicode[2221]:=16#64a4;
    unicode[2222]:=16#64a9;
    unicode[2223]:=16#64ac;
    unicode[2224]:=16#64ad;
    unicode[2225]:=16#64ae;
    unicode[2226]:=16#64b0;
    unicode[2227]:=16#64b5;
    unicode[2228]:=16#64b7;
    unicode[2229]:=16#64b8;
    unicode[2230]:=16#64ba;
    unicode[2231]:=16#64bc;
    unicode[2232]:=16#64c0;
    unicode[2233]:=16#64c2;
    unicode[2234]:=16#64c5;
    unicode[2235]:=16#64cd;
    unicode[2236]:=16#64ce;
    unicode[2237]:=16#64d0;
    unicode[2238]:=16#64d2;
    unicode[2239]:=16#64d7;
    unicode[2240]:=16#64d8;
    unicode[2241]:=16#64de;
    unicode[2242]:=16#64e2;
    unicode[2243]:=16#64e4;
    unicode[2244]:=16#64e6;
    unicode[2245]:=16#6500;
    unicode[2246]:=16#6509;
    unicode[2247]:=16#6512;
    unicode[2248]:=16#6518;
    unicode[2249]:=16#6525;
    unicode[2250]:=16#652b;
    unicode[2251]:=16#652e;
    unicode[2252]:=16#652f;
    unicode[2253]:=16#6534;
    unicode[2254]:=16#6535;
    unicode[2255]:=16#6536;
    unicode[2256]:=16#6538;
    unicode[2257]:=16#6539;
    unicode[2258]:=16#653b;
    unicode[2259]:=16#653e;
    unicode[2260]:=16#653f;
    unicode[2261]:=16#6545;
    unicode[2262]:=16#6548;
    unicode[2263]:=16#6549;
    unicode[2264]:=16#654c;
    unicode[2265]:=16#654f;
    unicode[2266]:=16#6551;
    unicode[2267]:=16#6555;
    unicode[2268]:=16#6556;
    unicode[2269]:=16#6559;
    unicode[2270]:=16#655b;
    unicode[2271]:=16#655d;
    unicode[2272]:=16#655e;
    unicode[2273]:=16#6562;
    unicode[2274]:=16#6563;
    unicode[2275]:=16#6566;
    unicode[2276]:=16#656b;
    unicode[2277]:=16#656c;
    unicode[2278]:=16#6570;
    unicode[2279]:=16#6572;
    unicode[2280]:=16#6574;
    unicode[2281]:=16#6577;
    unicode[2282]:=16#6587;
    unicode[2283]:=16#658b;
    unicode[2284]:=16#658c;
    unicode[2285]:=16#6590;
    unicode[2286]:=16#6591;
    unicode[2287]:=16#6593;
    unicode[2288]:=16#6597;
    unicode[2289]:=16#6599;
    unicode[2290]:=16#659b;
    unicode[2291]:=16#659c;
    unicode[2292]:=16#659f;
    unicode[2293]:=16#65a1;
    unicode[2294]:=16#65a4;
    unicode[2295]:=16#65a5;
    unicode[2296]:=16#65a7;
    unicode[2297]:=16#65a9;
    unicode[2298]:=16#65ab;
    unicode[2299]:=16#65ad;
    unicode[2300]:=16#65af;
    unicode[2301]:=16#65b0;
    unicode[2302]:=16#65b9;
    unicode[2303]:=16#65bc;
    unicode[2304]:=16#65bd;
    unicode[2305]:=16#65c1;
    unicode[2306]:=16#65c3;
    unicode[2307]:=16#65c4;
    unicode[2308]:=16#65c5;
    unicode[2309]:=16#65c6;
    unicode[2310]:=16#65cb;
    unicode[2311]:=16#65cc;
    unicode[2312]:=16#65ce;
    unicode[2313]:=16#65cf;
    unicode[2314]:=16#65d2;
    unicode[2315]:=16#65d6;
    unicode[2316]:=16#65d7;
    unicode[2317]:=16#65e0;
    unicode[2318]:=16#65e2;
    unicode[2319]:=16#65e5;
    unicode[2320]:=16#65e6;
    unicode[2321]:=16#65e7;
    unicode[2322]:=16#65e8;
    unicode[2323]:=16#65e9;
    unicode[2324]:=16#65ec;
    unicode[2325]:=16#65ed;
    unicode[2326]:=16#65ee;
    unicode[2327]:=16#65ef;
    unicode[2328]:=16#65f0;
    unicode[2329]:=16#65f1;
    unicode[2330]:=16#65f6;
    unicode[2331]:=16#65f7;
    unicode[2332]:=16#65fa;
    unicode[2333]:=16#6600;
    unicode[2334]:=16#6602;
    unicode[2335]:=16#6603;
    unicode[2336]:=16#6606;
    unicode[2337]:=16#660a;
    unicode[2338]:=16#660c;
    unicode[2339]:=16#660e;
    unicode[2340]:=16#660f;
    unicode[2341]:=16#6613;
    unicode[2342]:=16#6614;
    unicode[2343]:=16#6615;
    unicode[2344]:=16#6619;
    unicode[2345]:=16#661d;
    unicode[2346]:=16#661f;
    unicode[2347]:=16#6620;
    unicode[2348]:=16#6625;
    unicode[2349]:=16#6627;
    unicode[2350]:=16#6628;
    unicode[2351]:=16#662d;
    unicode[2352]:=16#662f;
    unicode[2353]:=16#6631;
    unicode[2354]:=16#6634;
    unicode[2355]:=16#6635;
    unicode[2356]:=16#6636;
    unicode[2357]:=16#663c;
    unicode[2358]:=16#663e;
    unicode[2359]:=16#6641;
    unicode[2360]:=16#6643;
    unicode[2361]:=16#664b;
    unicode[2362]:=16#664c;
    unicode[2363]:=16#664f;
    unicode[2364]:=16#6652;
    unicode[2365]:=16#6653;
    unicode[2366]:=16#6654;
    unicode[2367]:=16#6655;
    unicode[2368]:=16#6656;
    unicode[2369]:=16#6657;
    unicode[2370]:=16#665a;
    unicode[2371]:=16#665f;
    unicode[2372]:=16#6661;
    unicode[2373]:=16#6664;
    unicode[2374]:=16#6666;
    unicode[2375]:=16#6668;
    unicode[2376]:=16#666e;
    unicode[2377]:=16#666f;
    unicode[2378]:=16#6670;
    unicode[2379]:=16#6674;
    unicode[2380]:=16#6676;
    unicode[2381]:=16#6677;
    unicode[2382]:=16#667a;
    unicode[2383]:=16#667e;
    unicode[2384]:=16#6682;
    unicode[2385]:=16#6684;
    unicode[2386]:=16#6687;
    unicode[2387]:=16#668c;
    unicode[2388]:=16#6691;
    unicode[2389]:=16#6696;
    unicode[2390]:=16#6697;
    unicode[2391]:=16#669d;
    unicode[2392]:=16#66a7;
    unicode[2393]:=16#66a8;
    unicode[2394]:=16#66ae;
    unicode[2395]:=16#66b4;
    unicode[2396]:=16#66b9;
    unicode[2397]:=16#66be;
    unicode[2398]:=16#66d9;
    unicode[2399]:=16#66db;
    unicode[2400]:=16#66dc;
    unicode[2401]:=16#66dd;
    unicode[2402]:=16#66e6;
    unicode[2403]:=16#66e9;
    unicode[2404]:=16#66f0;
    unicode[2405]:=16#66f2;
    unicode[2406]:=16#66f3;
    unicode[2407]:=16#66f4;
    unicode[2408]:=16#66f7;
    unicode[2409]:=16#66f9;
    unicode[2410]:=16#66fc;
    unicode[2411]:=16#66fe;
    unicode[2412]:=16#66ff;
    unicode[2413]:=16#6700;
    unicode[2414]:=16#6708;
    unicode[2415]:=16#6709;
    unicode[2416]:=16#670a;
    unicode[2417]:=16#670b;
    unicode[2418]:=16#670d;
    unicode[2419]:=16#6710;
    unicode[2420]:=16#6714;
    unicode[2421]:=16#6715;
    unicode[2422]:=16#6717;
    unicode[2423]:=16#671b;
    unicode[2424]:=16#671d;
    unicode[2425]:=16#671f;
    unicode[2426]:=16#6726;
    unicode[2427]:=16#6728;
    unicode[2428]:=16#672a;
    unicode[2429]:=16#672b;
    unicode[2430]:=16#672c;
    unicode[2431]:=16#672d;
    unicode[2432]:=16#672f;
    unicode[2433]:=16#6731;
    unicode[2434]:=16#6734;
    unicode[2435]:=16#6735;
    unicode[2436]:=16#673a;
    unicode[2437]:=16#673d;
    unicode[2438]:=16#6740;
    unicode[2439]:=16#6742;
    unicode[2440]:=16#6743;
    unicode[2441]:=16#6746;
    unicode[2442]:=16#6748;
    unicode[2443]:=16#6749;
    unicode[2444]:=16#674c;
    unicode[2445]:=16#674e;
    unicode[2446]:=16#674f;
    unicode[2447]:=16#6750;
    unicode[2448]:=16#6751;
    unicode[2449]:=16#6753;
    unicode[2450]:=16#6756;
    unicode[2451]:=16#675c;
    unicode[2452]:=16#675e;
    unicode[2453]:=16#675f;
    unicode[2454]:=16#6760;
    unicode[2455]:=16#6761;
    unicode[2456]:=16#6765;
    unicode[2457]:=16#6768;
    unicode[2458]:=16#6769;
    unicode[2459]:=16#676a;
    unicode[2460]:=16#676d;
    unicode[2461]:=16#676f;
    unicode[2462]:=16#6770;
    unicode[2463]:=16#6772;
    unicode[2464]:=16#6773;
    unicode[2465]:=16#6775;
    unicode[2466]:=16#6777;
    unicode[2467]:=16#677c;
    unicode[2468]:=16#677e;
    unicode[2469]:=16#677f;
    unicode[2470]:=16#6781;
    unicode[2471]:=16#6784;
    unicode[2472]:=16#6787;
    unicode[2473]:=16#6789;
    unicode[2474]:=16#678b;
    unicode[2475]:=16#6790;
    unicode[2476]:=16#6795;
    unicode[2477]:=16#6797;
    unicode[2478]:=16#6798;
    unicode[2479]:=16#679a;
    unicode[2480]:=16#679c;
    unicode[2481]:=16#679d;
    unicode[2482]:=16#679e;
    unicode[2483]:=16#67a2;
    unicode[2484]:=16#67a3;
    unicode[2485]:=16#67a5;
    unicode[2486]:=16#67a7;
    unicode[2487]:=16#67a8;
    unicode[2488]:=16#67aa;
    unicode[2489]:=16#67ab;
    unicode[2490]:=16#67ad;
    unicode[2491]:=16#67af;
    unicode[2492]:=16#67b0;
    unicode[2493]:=16#67b3;
    unicode[2494]:=16#67b5;
    unicode[2495]:=16#67b6;
    unicode[2496]:=16#67b7;
    unicode[2497]:=16#67b8;
    unicode[2498]:=16#67c1;
    unicode[2499]:=16#67c3;
    unicode[2500]:=16#67c4;
    unicode[2501]:=16#67cf;
    unicode[2502]:=16#67d0;
    unicode[2503]:=16#67d1;
    unicode[2504]:=16#67d2;
    unicode[2505]:=16#67d3;
    unicode[2506]:=16#67d4;
    unicode[2507]:=16#67d8;
    unicode[2508]:=16#67d9;
    unicode[2509]:=16#67da;
    unicode[2510]:=16#67dc;
    unicode[2511]:=16#67dd;
    unicode[2512]:=16#67de;
    unicode[2513]:=16#67e0;
    unicode[2514]:=16#67e2;
    unicode[2515]:=16#67e5;
    unicode[2516]:=16#67e9;
    unicode[2517]:=16#67ec;
    unicode[2518]:=16#67ef;
    unicode[2519]:=16#67f0;
    unicode[2520]:=16#67f1;
    unicode[2521]:=16#67f3;
    unicode[2522]:=16#67f4;
    unicode[2523]:=16#67fd;
    unicode[2524]:=16#67ff;
    unicode[2525]:=16#6800;
    unicode[2526]:=16#6805;
    unicode[2527]:=16#6807;
    unicode[2528]:=16#6808;
    unicode[2529]:=16#6809;
    unicode[2530]:=16#680a;
    unicode[2531]:=16#680b;
    unicode[2532]:=16#680c;
    unicode[2533]:=16#680e;
    unicode[2534]:=16#680f;
    unicode[2535]:=16#6811;
    unicode[2536]:=16#6813;
    unicode[2537]:=16#6816;
    unicode[2538]:=16#6817;
    unicode[2539]:=16#681d;
    unicode[2540]:=16#6821;
    unicode[2541]:=16#6829;
    unicode[2542]:=16#682a;
    unicode[2543]:=16#6832;
    unicode[2544]:=16#6833;
    unicode[2545]:=16#6837;
    unicode[2546]:=16#6838;
    unicode[2547]:=16#6839;
    unicode[2548]:=16#683c;
    unicode[2549]:=16#683d;
    unicode[2550]:=16#683e;
    unicode[2551]:=16#6840;
    unicode[2552]:=16#6841;
    unicode[2553]:=16#6842;
    unicode[2554]:=16#6843;
    unicode[2555]:=16#6844;
    unicode[2556]:=16#6845;
    unicode[2557]:=16#6846;
    unicode[2558]:=16#6848;
    unicode[2559]:=16#6849;
    unicode[2560]:=16#684a;
    unicode[2561]:=16#684c;
    unicode[2562]:=16#684e;
    unicode[2563]:=16#6850;
    unicode[2564]:=16#6851;
    unicode[2565]:=16#6853;
    unicode[2566]:=16#6854;
    unicode[2567]:=16#6855;
    unicode[2568]:=16#6860;
    unicode[2569]:=16#6861;
    unicode[2570]:=16#6862;
    unicode[2571]:=16#6863;
    unicode[2572]:=16#6864;
    unicode[2573]:=16#6865;
    unicode[2574]:=16#6866;
    unicode[2575]:=16#6867;
    unicode[2576]:=16#6868;
    unicode[2577]:=16#6869;
    unicode[2578]:=16#686b;
    unicode[2579]:=16#6874;
    unicode[2580]:=16#6876;
    unicode[2581]:=16#6877;
    unicode[2582]:=16#6881;
    unicode[2583]:=16#6883;
    unicode[2584]:=16#6885;
    unicode[2585]:=16#6886;
    unicode[2586]:=16#688f;
    unicode[2587]:=16#6893;
    unicode[2588]:=16#6897;
    unicode[2589]:=16#68a2;
    unicode[2590]:=16#68a6;
    unicode[2591]:=16#68a7;
    unicode[2592]:=16#68a8;
    unicode[2593]:=16#68ad;
    unicode[2594]:=16#68af;
    unicode[2595]:=16#68b0;
    unicode[2596]:=16#68b3;
    unicode[2597]:=16#68b5;
    unicode[2598]:=16#68c0;
    unicode[2599]:=16#68c2;
    unicode[2600]:=16#68c9;
    unicode[2601]:=16#68cb;
    unicode[2602]:=16#68cd;
    unicode[2603]:=16#68d2;
    unicode[2604]:=16#68d5;
    unicode[2605]:=16#68d8;
    unicode[2606]:=16#68da;
    unicode[2607]:=16#68e0;
    unicode[2608]:=16#68e3;
    unicode[2609]:=16#68ee;
    unicode[2610]:=16#68f0;
    unicode[2611]:=16#68f1;
    unicode[2612]:=16#68f5;
    unicode[2613]:=16#68f9;
    unicode[2614]:=16#68fa;
    unicode[2615]:=16#68fc;
    unicode[2616]:=16#6901;
    unicode[2617]:=16#6905;
    unicode[2618]:=16#690b;
    unicode[2619]:=16#690d;
    unicode[2620]:=16#690e;
    unicode[2621]:=16#6910;
    unicode[2622]:=16#6912;
    unicode[2623]:=16#691f;
    unicode[2624]:=16#6920;
    unicode[2625]:=16#6924;
    unicode[2626]:=16#692d;
    unicode[2627]:=16#6930;
    unicode[2628]:=16#6934;
    unicode[2629]:=16#6939;
    unicode[2630]:=16#693d;
    unicode[2631]:=16#693f;
    unicode[2632]:=16#6942;
    unicode[2633]:=16#6954;
    unicode[2634]:=16#6957;
    unicode[2635]:=16#695a;
    unicode[2636]:=16#695d;
    unicode[2637]:=16#695e;
    unicode[2638]:=16#6960;
    unicode[2639]:=16#6963;
    unicode[2640]:=16#6966;
    unicode[2641]:=16#696b;
    unicode[2642]:=16#696e;
    unicode[2643]:=16#6971;
    unicode[2644]:=16#6977;
    unicode[2645]:=16#6978;
    unicode[2646]:=16#6979;
    unicode[2647]:=16#697c;
    unicode[2648]:=16#6980;
    unicode[2649]:=16#6982;
    unicode[2650]:=16#6984;
    unicode[2651]:=16#6986;
    unicode[2652]:=16#6987;
    unicode[2653]:=16#6988;
    unicode[2654]:=16#6989;
    unicode[2655]:=16#698d;
    unicode[2656]:=16#6994;
    unicode[2657]:=16#6995;
    unicode[2658]:=16#6998;
    unicode[2659]:=16#699b;
    unicode[2660]:=16#699c;
    unicode[2661]:=16#69a7;
    unicode[2662]:=16#69a8;
    unicode[2663]:=16#69ab;
    unicode[2664]:=16#69ad;
    unicode[2665]:=16#69b1;
    unicode[2666]:=16#69b4;
    unicode[2667]:=16#69b7;
    unicode[2668]:=16#69bb;
    unicode[2669]:=16#69c1;
    unicode[2670]:=16#69ca;
    unicode[2671]:=16#69cc;
    unicode[2672]:=16#69ce;
    unicode[2673]:=16#69d0;
    unicode[2674]:=16#69d4;
    unicode[2675]:=16#69db;
    unicode[2676]:=16#69df;
    unicode[2677]:=16#69e0;
    unicode[2678]:=16#69ed;
    unicode[2679]:=16#69f2;
    unicode[2680]:=16#69fd;
    unicode[2681]:=16#69ff;
    unicode[2682]:=16#6a0a;
    unicode[2683]:=16#6a17;
    unicode[2684]:=16#6a18;
    unicode[2685]:=16#6a1f;
    unicode[2686]:=16#6a21;
    unicode[2687]:=16#6a28;
    unicode[2688]:=16#6a2a;
    unicode[2689]:=16#6a2f;
    unicode[2690]:=16#6a31;
    unicode[2691]:=16#6a35;
    unicode[2692]:=16#6a3d;
    unicode[2693]:=16#6a3e;
    unicode[2694]:=16#6a44;
    unicode[2695]:=16#6a47;
    unicode[2696]:=16#6a50;
    unicode[2697]:=16#6a58;
    unicode[2698]:=16#6a59;
    unicode[2699]:=16#6a5b;
    unicode[2700]:=16#6a61;
    unicode[2701]:=16#6a65;
    unicode[2702]:=16#6a71;
    unicode[2703]:=16#6a79;
    unicode[2704]:=16#6a7c;
    unicode[2705]:=16#6a80;
    unicode[2706]:=16#6a84;
    unicode[2707]:=16#6a8e;
    unicode[2708]:=16#6a90;
    unicode[2709]:=16#6a91;
    unicode[2710]:=16#6a97;
    unicode[2711]:=16#6aa0;
    unicode[2712]:=16#6aa9;
    unicode[2713]:=16#6aab;
    unicode[2714]:=16#6aac;
    unicode[2715]:=16#6b20;
    unicode[2716]:=16#6b21;
    unicode[2717]:=16#6b22;
    unicode[2718]:=16#6b23;
    unicode[2719]:=16#6b24;
    unicode[2720]:=16#6b27;
    unicode[2721]:=16#6b32;
    unicode[2722]:=16#6b37;
    unicode[2723]:=16#6b39;
    unicode[2724]:=16#6b3a;
    unicode[2725]:=16#6b3e;
    unicode[2726]:=16#6b43;
    unicode[2727]:=16#6b46;
    unicode[2728]:=16#6b47;
    unicode[2729]:=16#6b49;
    unicode[2730]:=16#6b4c;
    unicode[2731]:=16#6b59;
    unicode[2732]:=16#6b62;
    unicode[2733]:=16#6b63;
    unicode[2734]:=16#6b64;
    unicode[2735]:=16#6b65;
    unicode[2736]:=16#6b66;
    unicode[2737]:=16#6b67;
    unicode[2738]:=16#6b6a;
    unicode[2739]:=16#6b79;
    unicode[2740]:=16#6b7b;
    unicode[2741]:=16#6b7c;
    unicode[2742]:=16#6b81;
    unicode[2743]:=16#6b82;
    unicode[2744]:=16#6b83;
    unicode[2745]:=16#6b84;
    unicode[2746]:=16#6b86;
    unicode[2747]:=16#6b87;
    unicode[2748]:=16#6b89;
    unicode[2749]:=16#6b8a;
    unicode[2750]:=16#6b8b;
    unicode[2751]:=16#6b8d;
    unicode[2752]:=16#6b92;
    unicode[2753]:=16#6b93;
    unicode[2754]:=16#6b96;
    unicode[2755]:=16#6b9a;
    unicode[2756]:=16#6b9b;
    unicode[2757]:=16#6ba1;
    unicode[2758]:=16#6baa;
    unicode[2759]:=16#6bb3;
    unicode[2760]:=16#6bb4;
    unicode[2761]:=16#6bb5;
    unicode[2762]:=16#6bb7;
    unicode[2763]:=16#6bbf;
    unicode[2764]:=16#6bc1;
    unicode[2765]:=16#6bc2;
    unicode[2766]:=16#6bc5;
    unicode[2767]:=16#6bcb;
    unicode[2768]:=16#6bcd;
    unicode[2769]:=16#6bcf;
    unicode[2770]:=16#6bd2;
    unicode[2771]:=16#6bd3;
    unicode[2772]:=16#6bd4;
    unicode[2773]:=16#6bd5;
    unicode[2774]:=16#6bd6;
    unicode[2775]:=16#6bd7;
    unicode[2776]:=16#6bd9;
    unicode[2777]:=16#6bdb;
    unicode[2778]:=16#6be1;
    unicode[2779]:=16#6bea;
    unicode[2780]:=16#6beb;
    unicode[2781]:=16#6bef;
    unicode[2782]:=16#6bf3;
    unicode[2783]:=16#6bf5;
    unicode[2784]:=16#6bf9;
    unicode[2785]:=16#6bfd;
    unicode[2786]:=16#6c05;
    unicode[2787]:=16#6c06;
    unicode[2788]:=16#6c07;
    unicode[2789]:=16#6c0d;
    unicode[2790]:=16#6c0f;
    unicode[2791]:=16#6c10;
    unicode[2792]:=16#6c11;
    unicode[2793]:=16#6c13;
    unicode[2794]:=16#6c14;
    unicode[2795]:=16#6c15;
    unicode[2796]:=16#6c16;
    unicode[2797]:=16#6c18;
    unicode[2798]:=16#6c19;
    unicode[2799]:=16#6c1a;
    unicode[2800]:=16#6c1b;
    unicode[2801]:=16#6c1f;
    unicode[2802]:=16#6c21;
    unicode[2803]:=16#6c22;
    unicode[2804]:=16#6c24;
    unicode[2805]:=16#6c26;
    unicode[2806]:=16#6c27;
    unicode[2807]:=16#6c28;
    unicode[2808]:=16#6c29;
    unicode[2809]:=16#6c2a;
    unicode[2810]:=16#6c2e;
    unicode[2811]:=16#6c2f;
    unicode[2812]:=16#6c30;
    unicode[2813]:=16#6c32;
    unicode[2814]:=16#6c34;
    unicode[2815]:=16#6c35;
    unicode[2816]:=16#6c38;
    unicode[2817]:=16#6c3d;
    unicode[2818]:=16#6c40;
    unicode[2819]:=16#6c41;
    unicode[2820]:=16#6c42;
    unicode[2821]:=16#6c46;
    unicode[2822]:=16#6c47;
    unicode[2823]:=16#6c49;
    unicode[2824]:=16#6c4a;
    unicode[2825]:=16#6c50;
    unicode[2826]:=16#6c54;
    unicode[2827]:=16#6c55;
    unicode[2828]:=16#6c57;
    unicode[2829]:=16#6c5b;
    unicode[2830]:=16#6c5c;
    unicode[2831]:=16#6c5d;
    unicode[2832]:=16#6c5e;
    unicode[2833]:=16#6c5f;
    unicode[2834]:=16#6c60;
    unicode[2835]:=16#6c61;
    unicode[2836]:=16#6c64;
    unicode[2837]:=16#6c68;
    unicode[2838]:=16#6c69;
    unicode[2839]:=16#6c6a;
    unicode[2840]:=16#6c70;
    unicode[2841]:=16#6c72;
    unicode[2842]:=16#6c74;
    unicode[2843]:=16#6c76;
    unicode[2844]:=16#6c79;
    unicode[2845]:=16#6c7d;
    unicode[2846]:=16#6c7e;
    unicode[2847]:=16#6c81;
    unicode[2848]:=16#6c82;
    unicode[2849]:=16#6c83;
    unicode[2850]:=16#6c85;
    unicode[2851]:=16#6c86;
    unicode[2852]:=16#6c88;
    unicode[2853]:=16#6c89;
    unicode[2854]:=16#6c8c;
    unicode[2855]:=16#6c8f;
    unicode[2856]:=16#6c90;
    unicode[2857]:=16#6c93;
    unicode[2858]:=16#6c94;
    unicode[2859]:=16#6c99;
    unicode[2860]:=16#6c9b;
    unicode[2861]:=16#6c9f;
    unicode[2862]:=16#6ca1;
    unicode[2863]:=16#6ca3;
    unicode[2864]:=16#6ca4;
    unicode[2865]:=16#6ca5;
    unicode[2866]:=16#6ca6;
    unicode[2867]:=16#6ca7;
    unicode[2868]:=16#6ca9;
    unicode[2869]:=16#6caa;
    unicode[2870]:=16#6cab;
    unicode[2871]:=16#6cad;
    unicode[2872]:=16#6cae;
    unicode[2873]:=16#6cb1;
    unicode[2874]:=16#6cb2;
    unicode[2875]:=16#6cb3;
    unicode[2876]:=16#6cb8;
    unicode[2877]:=16#6cb9;
    unicode[2878]:=16#6cbb;
    unicode[2879]:=16#6cbc;
    unicode[2880]:=16#6cbd;
    unicode[2881]:=16#6cbe;
    unicode[2882]:=16#6cbf;
    unicode[2883]:=16#6cc4;
    unicode[2884]:=16#6cc5;
    unicode[2885]:=16#6cc9;
    unicode[2886]:=16#6cca;
    unicode[2887]:=16#6ccc;
    unicode[2888]:=16#6cd0;
    unicode[2889]:=16#6cd3;
    unicode[2890]:=16#6cd4;
    unicode[2891]:=16#6cd5;
    unicode[2892]:=16#6cd6;
    unicode[2893]:=16#6cd7;
    unicode[2894]:=16#6cdb;
    unicode[2895]:=16#6cde;
    unicode[2896]:=16#6ce0;
    unicode[2897]:=16#6ce1;
    unicode[2898]:=16#6ce2;
    unicode[2899]:=16#6ce3;
    unicode[2900]:=16#6ce5;
    unicode[2901]:=16#6ce8;
    unicode[2902]:=16#6cea;
    unicode[2903]:=16#6ceb;
    unicode[2904]:=16#6cee;
    unicode[2905]:=16#6cef;
    unicode[2906]:=16#6cf0;
    unicode[2907]:=16#6cf1;
    unicode[2908]:=16#6cf3;
    unicode[2909]:=16#6cf5;
    unicode[2910]:=16#6cf6;
    unicode[2911]:=16#6cf7;
    unicode[2912]:=16#6cf8;
    unicode[2913]:=16#6cfa;
    unicode[2914]:=16#6cfb;
    unicode[2915]:=16#6cfc;
    unicode[2916]:=16#6cfd;
    unicode[2917]:=16#6cfe;
    unicode[2918]:=16#6d01;
    unicode[2919]:=16#6d04;
    unicode[2920]:=16#6d07;
    unicode[2921]:=16#6d0b;
    unicode[2922]:=16#6d0c;
    unicode[2923]:=16#6d0e;
    unicode[2924]:=16#6d12;
    unicode[2925]:=16#6d17;
    unicode[2926]:=16#6d19;
    unicode[2927]:=16#6d1a;
    unicode[2928]:=16#6d1b;
    unicode[2929]:=16#6d1e;
    unicode[2930]:=16#6d25;
    unicode[2931]:=16#6d27;
    unicode[2932]:=16#6d2a;
    unicode[2933]:=16#6d2b;
    unicode[2934]:=16#6d2e;
    unicode[2935]:=16#6d31;
    unicode[2936]:=16#6d32;
    unicode[2937]:=16#6d33;
    unicode[2938]:=16#6d35;
    unicode[2939]:=16#6d39;
    unicode[2940]:=16#6d3b;
    unicode[2941]:=16#6d3c;
    unicode[2942]:=16#6d3d;
    unicode[2943]:=16#6d3e;
    unicode[2944]:=16#6d41;
    unicode[2945]:=16#6d43;
    unicode[2946]:=16#6d45;
    unicode[2947]:=16#6d46;
    unicode[2948]:=16#6d47;
    unicode[2949]:=16#6d48;
    unicode[2950]:=16#6d4a;
    unicode[2951]:=16#6d4b;
    unicode[2952]:=16#6d4d;
    unicode[2953]:=16#6d4e;
    unicode[2954]:=16#6d4f;
    unicode[2955]:=16#6d51;
    unicode[2956]:=16#6d52;
    unicode[2957]:=16#6d53;
    unicode[2958]:=16#6d54;
    unicode[2959]:=16#6d59;
    unicode[2960]:=16#6d5a;
    unicode[2961]:=16#6d5c;
    unicode[2962]:=16#6d5e;
    unicode[2963]:=16#6d60;
    unicode[2964]:=16#6d63;
    unicode[2965]:=16#6d66;
    unicode[2966]:=16#6d69;
    unicode[2967]:=16#6d6a;
    unicode[2968]:=16#6d6e;
    unicode[2969]:=16#6d6f;
    unicode[2970]:=16#6d74;
    unicode[2971]:=16#6d77;
    unicode[2972]:=16#6d78;
    unicode[2973]:=16#6d7c;
    unicode[2974]:=16#6d82;
    unicode[2975]:=16#6d85;
    unicode[2976]:=16#6d88;
    unicode[2977]:=16#6d89;
    unicode[2978]:=16#6d8c;
    unicode[2979]:=16#6d8e;
    unicode[2980]:=16#6d91;
    unicode[2981]:=16#6d93;
    unicode[2982]:=16#6d94;
    unicode[2983]:=16#6d95;
    unicode[2984]:=16#6d9b;
    unicode[2985]:=16#6d9d;
    unicode[2986]:=16#6d9e;
    unicode[2987]:=16#6d9f;
    unicode[2988]:=16#6da0;
    unicode[2989]:=16#6da1;
    unicode[2990]:=16#6da3;
    unicode[2991]:=16#6da4;
    unicode[2992]:=16#6da6;
    unicode[2993]:=16#6da7;
    unicode[2994]:=16#6da8;
    unicode[2995]:=16#6da9;
    unicode[2996]:=16#6daa;
    unicode[2997]:=16#6dab;
    unicode[2998]:=16#6dae;
    unicode[2999]:=16#6daf;            //unicode码 2000-2999
END_IF;
(* Rung 7 *)
IF P_On THEN
    unicode[3000]:=16#6db2;
    unicode[3001]:=16#6db5;
    unicode[3002]:=16#6db8;
    unicode[3003]:=16#6dbf;
    unicode[3004]:=16#6dc0;
    unicode[3005]:=16#6dc4;
    unicode[3006]:=16#6dc5;
    unicode[3007]:=16#6dc6;
    unicode[3008]:=16#6dc7;
    unicode[3009]:=16#6dcb;
    unicode[3010]:=16#6dcc;
    unicode[3011]:=16#6dd1;
    unicode[3012]:=16#6dd6;
    unicode[3013]:=16#6dd8;
    unicode[3014]:=16#6dd9;
    unicode[3015]:=16#6ddd;
    unicode[3016]:=16#6dde;
    unicode[3017]:=16#6de0;
    unicode[3018]:=16#6de1;
    unicode[3019]:=16#6de4;
    unicode[3020]:=16#6de6;
    unicode[3021]:=16#6deb;
    unicode[3022]:=16#6dec;
    unicode[3023]:=16#6dee;
    unicode[3024]:=16#6df1;
    unicode[3025]:=16#6df3;
    unicode[3026]:=16#6df7;
    unicode[3027]:=16#6df9;
    unicode[3028]:=16#6dfb;
    unicode[3029]:=16#6dfc;
    unicode[3030]:=16#6e05;
    unicode[3031]:=16#6e0a;
    unicode[3032]:=16#6e0c;
    unicode[3033]:=16#6e0d;
    unicode[3034]:=16#6e0e;
    unicode[3035]:=16#6e10;
    unicode[3036]:=16#6e11;
    unicode[3037]:=16#6e14;
    unicode[3038]:=16#6e16;
    unicode[3039]:=16#6e17;
    unicode[3040]:=16#6e1a;
    unicode[3041]:=16#6e1d;
    unicode[3042]:=16#6e20;
    unicode[3043]:=16#6e21;
    unicode[3044]:=16#6e23;
    unicode[3045]:=16#6e24;
    unicode[3046]:=16#6e25;
    unicode[3047]:=16#6e29;
    unicode[3048]:=16#6e2b;
    unicode[3049]:=16#6e2d;
    unicode[3050]:=16#6e2f;
    unicode[3051]:=16#6e32;
    unicode[3052]:=16#6e34;
    unicode[3053]:=16#6e38;
    unicode[3054]:=16#6e3a;
    unicode[3055]:=16#6e43;
    unicode[3056]:=16#6e44;
    unicode[3057]:=16#6e4d;
    unicode[3058]:=16#6e4e;
    unicode[3059]:=16#6e53;
    unicode[3060]:=16#6e54;
    unicode[3061]:=16#6e56;
    unicode[3062]:=16#6e58;
    unicode[3063]:=16#6e5b;
    unicode[3064]:=16#6e5f;
    unicode[3065]:=16#6e6b;
    unicode[3066]:=16#6e6e;
    unicode[3067]:=16#6e7e;
    unicode[3068]:=16#6e7f;
    unicode[3069]:=16#6e83;
    unicode[3070]:=16#6e85;
    unicode[3071]:=16#6e86;
    unicode[3072]:=16#6e89;
    unicode[3073]:=16#6e8f;
    unicode[3074]:=16#6e90;
    unicode[3075]:=16#6e98;
    unicode[3076]:=16#6e9c;
    unicode[3077]:=16#6e9f;
    unicode[3078]:=16#6ea2;
    unicode[3079]:=16#6ea5;
    unicode[3080]:=16#6ea7;
    unicode[3081]:=16#6eaa;
    unicode[3082]:=16#6eaf;
    unicode[3083]:=16#6eb1;
    unicode[3084]:=16#6eb2;
    unicode[3085]:=16#6eb4;
    unicode[3086]:=16#6eb6;
    unicode[3087]:=16#6eb7;
    unicode[3088]:=16#6eba;
    unicode[3089]:=16#6ebb;
    unicode[3090]:=16#6ebd;
    unicode[3091]:=16#6ec1;
    unicode[3092]:=16#6ec2;
    unicode[3093]:=16#6ec7;
    unicode[3094]:=16#6ecb;
    unicode[3095]:=16#6ecf;
    unicode[3096]:=16#6ed1;
    unicode[3097]:=16#6ed3;
    unicode[3098]:=16#6ed4;
    unicode[3099]:=16#6ed5;
    unicode[3100]:=16#6ed7;
    unicode[3101]:=16#6eda;
    unicode[3102]:=16#6ede;
    unicode[3103]:=16#6edf;
    unicode[3104]:=16#6ee0;
    unicode[3105]:=16#6ee1;
    unicode[3106]:=16#6ee2;
    unicode[3107]:=16#6ee4;
    unicode[3108]:=16#6ee5;
    unicode[3109]:=16#6ee6;
    unicode[3110]:=16#6ee8;
    unicode[3111]:=16#6ee9;
    unicode[3112]:=16#6ef4;
    unicode[3113]:=16#6ef9;
    unicode[3114]:=16#6f02;
    unicode[3115]:=16#6f06;
    unicode[3116]:=16#6f09;
    unicode[3117]:=16#6f0f;
    unicode[3118]:=16#6f13;
    unicode[3119]:=16#6f14;
    unicode[3120]:=16#6f15;
    unicode[3121]:=16#6f20;
    unicode[3122]:=16#6f24;
    unicode[3123]:=16#6f29;
    unicode[3124]:=16#6f2a;
    unicode[3125]:=16#6f2b;
    unicode[3126]:=16#6f2d;
    unicode[3127]:=16#6f2f;
    unicode[3128]:=16#6f31;
    unicode[3129]:=16#6f33;
    unicode[3130]:=16#6f36;
    unicode[3131]:=16#6f3e;
    unicode[3132]:=16#6f46;
    unicode[3133]:=16#6f47;
    unicode[3134]:=16#6f4b;
    unicode[3135]:=16#6f4d;
    unicode[3136]:=16#6f58;
    unicode[3137]:=16#6f5c;
    unicode[3138]:=16#6f5e;
    unicode[3139]:=16#6f62;
    unicode[3140]:=16#6f66;
    unicode[3141]:=16#6f6d;
    unicode[3142]:=16#6f6e;
    unicode[3143]:=16#6f72;
    unicode[3144]:=16#6f74;
    unicode[3145]:=16#6f78;
    unicode[3146]:=16#6f7a;
    unicode[3147]:=16#6f7c;
    unicode[3148]:=16#6f84;
    unicode[3149]:=16#6f88;
    unicode[3150]:=16#6f89;
    unicode[3151]:=16#6f8c;
    unicode[3152]:=16#6f8d;
    unicode[3153]:=16#6f8e;
    unicode[3154]:=16#6f9c;
    unicode[3155]:=16#6fa1;
    unicode[3156]:=16#6fa7;
    unicode[3157]:=16#6fb3;
    unicode[3158]:=16#6fb6;
    unicode[3159]:=16#6fb9;
    unicode[3160]:=16#6fc0;
    unicode[3161]:=16#6fc2;
    unicode[3162]:=16#6fc9;
    unicode[3163]:=16#6fd1;
    unicode[3164]:=16#6fd2;
    unicode[3165]:=16#6fde;
    unicode[3166]:=16#6fe0;
    unicode[3167]:=16#6fe1;
    unicode[3168]:=16#6fee;
    unicode[3169]:=16#6fef;
    unicode[3170]:=16#7011;
    unicode[3171]:=16#701a;
    unicode[3172]:=16#701b;
    unicode[3173]:=16#7023;
    unicode[3174]:=16#7035;
    unicode[3175]:=16#7039;
    unicode[3176]:=16#704c;
    unicode[3177]:=16#704f;
    unicode[3178]:=16#705e;
    unicode[3179]:=16#706b;
    unicode[3180]:=16#706c;
    unicode[3181]:=16#706d;
    unicode[3182]:=16#706f;
    unicode[3183]:=16#7070;
    unicode[3184]:=16#7075;
    unicode[3185]:=16#7076;
    unicode[3186]:=16#7078;
    unicode[3187]:=16#707c;
    unicode[3188]:=16#707e;
    unicode[3189]:=16#707f;
    unicode[3190]:=16#7080;
    unicode[3191]:=16#7085;
    unicode[3192]:=16#7089;
    unicode[3193]:=16#708a;
    unicode[3194]:=16#708e;
    unicode[3195]:=16#7092;
    unicode[3196]:=16#7094;
    unicode[3197]:=16#7095;
    unicode[3198]:=16#7096;
    unicode[3199]:=16#7099;
    unicode[3200]:=16#709c;
    unicode[3201]:=16#709d;
    unicode[3202]:=16#70ab;
    unicode[3203]:=16#70ac;
    unicode[3204]:=16#70ad;
    unicode[3205]:=16#70ae;
    unicode[3206]:=16#70af;
    unicode[3207]:=16#70b1;
    unicode[3208]:=16#70b3;
    unicode[3209]:=16#70b7;
    unicode[3210]:=16#70b8;
    unicode[3211]:=16#70b9;
    unicode[3212]:=16#70bb;
    unicode[3213]:=16#70bc;
    unicode[3214]:=16#70bd;
    unicode[3215]:=16#70c0;
    unicode[3216]:=16#70c1;
    unicode[3217]:=16#70c2;
    unicode[3218]:=16#70c3;
    unicode[3219]:=16#70c8;
    unicode[3220]:=16#70ca;
    unicode[3221]:=16#70d8;
    unicode[3222]:=16#70d9;
    unicode[3223]:=16#70db;
    unicode[3224]:=16#70df;
    unicode[3225]:=16#70e4;
    unicode[3226]:=16#70e6;
    unicode[3227]:=16#70e7;
    unicode[3228]:=16#70e8;
    unicode[3229]:=16#70e9;
    unicode[3230]:=16#70eb;
    unicode[3231]:=16#70ec;
    unicode[3232]:=16#70ed;
    unicode[3233]:=16#70ef;
    unicode[3234]:=16#70f7;
    unicode[3235]:=16#70f9;
    unicode[3236]:=16#70fd;
    unicode[3237]:=16#7109;
    unicode[3238]:=16#710a;
    unicode[3239]:=16#7110;
    unicode[3240]:=16#7113;
    unicode[3241]:=16#7115;
    unicode[3242]:=16#7116;
    unicode[3243]:=16#7118;
    unicode[3244]:=16#7119;
    unicode[3245]:=16#711a;
    unicode[3246]:=16#7126;
    unicode[3247]:=16#712f;
    unicode[3248]:=16#7130;
    unicode[3249]:=16#7131;
    unicode[3250]:=16#7136;
    unicode[3251]:=16#7145;
    unicode[3252]:=16#714a;
    unicode[3253]:=16#714c;
    unicode[3254]:=16#714e;
    unicode[3255]:=16#715c;
    unicode[3256]:=16#715e;
    unicode[3257]:=16#7164;
    unicode[3258]:=16#7166;
    unicode[3259]:=16#7167;
    unicode[3260]:=16#7168;
    unicode[3261]:=16#716e;
    unicode[3262]:=16#7172;
    unicode[3263]:=16#7173;
    unicode[3264]:=16#7178;
    unicode[3265]:=16#717a;
    unicode[3266]:=16#717d;
    unicode[3267]:=16#7184;
    unicode[3268]:=16#718a;
    unicode[3269]:=16#718f;
    unicode[3270]:=16#7194;
    unicode[3271]:=16#7198;
    unicode[3272]:=16#7199;
    unicode[3273]:=16#719f;
    unicode[3274]:=16#71a0;
    unicode[3275]:=16#71a8;
    unicode[3276]:=16#71ac;
    unicode[3277]:=16#71b3;
    unicode[3278]:=16#71b5;
    unicode[3279]:=16#71b9;
    unicode[3280]:=16#71c3;
    unicode[3281]:=16#71ce;
    unicode[3282]:=16#71d4;
    unicode[3283]:=16#71d5;
    unicode[3284]:=16#71e0;
    unicode[3285]:=16#71e5;
    unicode[3286]:=16#71e7;
    unicode[3287]:=16#71ee;
    unicode[3288]:=16#71f9;
    unicode[3289]:=16#7206;
    unicode[3290]:=16#721d;
    unicode[3291]:=16#7228;
    unicode[3292]:=16#722a;
    unicode[3293]:=16#722c;
    unicode[3294]:=16#7230;
    unicode[3295]:=16#7231;
    unicode[3296]:=16#7235;
    unicode[3297]:=16#7236;
    unicode[3298]:=16#7237;
    unicode[3299]:=16#7238;
    unicode[3300]:=16#7239;
    unicode[3301]:=16#723b;
    unicode[3302]:=16#723d;
    unicode[3303]:=16#723f;
    unicode[3304]:=16#7247;
    unicode[3305]:=16#7248;
    unicode[3306]:=16#724c;
    unicode[3307]:=16#724d;
    unicode[3308]:=16#7252;
    unicode[3309]:=16#7256;
    unicode[3310]:=16#7259;
    unicode[3311]:=16#725b;
    unicode[3312]:=16#725d;
    unicode[3313]:=16#725f;
    unicode[3314]:=16#7261;
    unicode[3315]:=16#7262;
    unicode[3316]:=16#7266;
    unicode[3317]:=16#7267;
    unicode[3318]:=16#7269;
    unicode[3319]:=16#726e;
    unicode[3320]:=16#726f;
    unicode[3321]:=16#7272;
    unicode[3322]:=16#7275;
    unicode[3323]:=16#7279;
    unicode[3324]:=16#727a;
    unicode[3325]:=16#727e;
    unicode[3326]:=16#727f;
    unicode[3327]:=16#7280;
    unicode[3328]:=16#7281;
    unicode[3329]:=16#7284;
    unicode[3330]:=16#728a;
    unicode[3331]:=16#728b;
    unicode[3332]:=16#728d;
    unicode[3333]:=16#728f;
    unicode[3334]:=16#7292;
    unicode[3335]:=16#729f;
    unicode[3336]:=16#72ac;
    unicode[3337]:=16#72ad;
    unicode[3338]:=16#72af;
    unicode[3339]:=16#72b0;
    unicode[3340]:=16#72b4;
    unicode[3341]:=16#72b6;
    unicode[3342]:=16#72b7;
    unicode[3343]:=16#72b8;
    unicode[3344]:=16#72b9;
    unicode[3345]:=16#72c1;
    unicode[3346]:=16#72c2;
    unicode[3347]:=16#72c3;
    unicode[3348]:=16#72c4;
    unicode[3349]:=16#72c8;
    unicode[3350]:=16#72cd;
    unicode[3351]:=16#72ce;
    unicode[3352]:=16#72d0;
    unicode[3353]:=16#72d2;
    unicode[3354]:=16#72d7;
    unicode[3355]:=16#72d9;
    unicode[3356]:=16#72de;
    unicode[3357]:=16#72e0;
    unicode[3358]:=16#72e1;
    unicode[3359]:=16#72e8;
    unicode[3360]:=16#72e9;
    unicode[3361]:=16#72ec;
    unicode[3362]:=16#72ed;
    unicode[3363]:=16#72ee;
    unicode[3364]:=16#72ef;
    unicode[3365]:=16#72f0;
    unicode[3366]:=16#72f1;
    unicode[3367]:=16#72f2;
    unicode[3368]:=16#72f3;
    unicode[3369]:=16#72f4;
    unicode[3370]:=16#72f7;
    unicode[3371]:=16#72f8;
    unicode[3372]:=16#72fa;
    unicode[3373]:=16#72fb;
    unicode[3374]:=16#72fc;
    unicode[3375]:=16#7301;
    unicode[3376]:=16#7303;
    unicode[3377]:=16#730a;
    unicode[3378]:=16#730e;
    unicode[3379]:=16#7313;
    unicode[3380]:=16#7315;
    unicode[3381]:=16#7316;
    unicode[3382]:=16#7317;
    unicode[3383]:=16#731b;
    unicode[3384]:=16#731c;
    unicode[3385]:=16#731d;
    unicode[3386]:=16#731e;
    unicode[3387]:=16#7321;
    unicode[3388]:=16#7322;
    unicode[3389]:=16#7325;
    unicode[3390]:=16#7329;
    unicode[3391]:=16#732a;
    unicode[3392]:=16#732b;
    unicode[3393]:=16#732c;
    unicode[3394]:=16#732e;
    unicode[3395]:=16#7331;
    unicode[3396]:=16#7334;
    unicode[3397]:=16#7337;
    unicode[3398]:=16#7338;
    unicode[3399]:=16#7339;
    unicode[3400]:=16#733e;
    unicode[3401]:=16#733f;
    unicode[3402]:=16#734d;
    unicode[3403]:=16#7350;
    unicode[3404]:=16#7352;
    unicode[3405]:=16#7357;
    unicode[3406]:=16#7360;
    unicode[3407]:=16#736c;
    unicode[3408]:=16#736d;
    unicode[3409]:=16#736f;
    unicode[3410]:=16#737e;
    unicode[3411]:=16#7384;
    unicode[3412]:=16#7387;
    unicode[3413]:=16#7389;
    unicode[3414]:=16#738b;
    unicode[3415]:=16#738e;
    unicode[3416]:=16#7391;
    unicode[3417]:=16#7396;
    unicode[3418]:=16#739b;
    unicode[3419]:=16#739f;
    unicode[3420]:=16#73a2;
    unicode[3421]:=16#73a9;
    unicode[3422]:=16#73ab;
    unicode[3423]:=16#73ae;
    unicode[3424]:=16#73af;
    unicode[3425]:=16#73b0;
    unicode[3426]:=16#73b2;
    unicode[3427]:=16#73b3;
    unicode[3428]:=16#73b7;
    unicode[3429]:=16#73ba;
    unicode[3430]:=16#73bb;
    unicode[3431]:=16#73c0;
    unicode[3432]:=16#73c2;
    unicode[3433]:=16#73c8;
    unicode[3434]:=16#73c9;
    unicode[3435]:=16#73ca;
    unicode[3436]:=16#73cd;
    unicode[3437]:=16#73cf;
    unicode[3438]:=16#73d0;
    unicode[3439]:=16#73d1;
    unicode[3440]:=16#73d9;
    unicode[3441]:=16#73de;
    unicode[3442]:=16#73e0;
    unicode[3443]:=16#73e5;
    unicode[3444]:=16#73e7;
    unicode[3445]:=16#73e9;
    unicode[3446]:=16#73ed;
    unicode[3447]:=16#73f2;
    unicode[3448]:=16#7403;
    unicode[3449]:=16#7405;
    unicode[3450]:=16#7406;
    unicode[3451]:=16#7409;
    unicode[3452]:=16#740a;
    unicode[3453]:=16#740f;
    unicode[3454]:=16#7410;
    unicode[3455]:=16#741a;
    unicode[3456]:=16#741b;
    unicode[3457]:=16#7422;
    unicode[3458]:=16#7425;
    unicode[3459]:=16#7426;
    unicode[3460]:=16#7428;
    unicode[3461]:=16#742a;
    unicode[3462]:=16#742c;
    unicode[3463]:=16#742e;
    unicode[3464]:=16#7430;
    unicode[3465]:=16#7433;
    unicode[3466]:=16#7434;
    unicode[3467]:=16#7435;
    unicode[3468]:=16#7436;
    unicode[3469]:=16#743c;
    unicode[3470]:=16#7441;
    unicode[3471]:=16#7455;
    unicode[3472]:=16#7457;
    unicode[3473]:=16#7459;
    unicode[3474]:=16#745a;
    unicode[3475]:=16#745b;
    unicode[3476]:=16#745c;
    unicode[3477]:=16#745e;
    unicode[3478]:=16#745f;
    unicode[3479]:=16#746d;
    unicode[3480]:=16#7470;
    unicode[3481]:=16#7476;
    unicode[3482]:=16#7477;
    unicode[3483]:=16#747e;
    unicode[3484]:=16#7480;
    unicode[3485]:=16#7481;
    unicode[3486]:=16#7483;
    unicode[3487]:=16#7487;
    unicode[3488]:=16#748b;
    unicode[3489]:=16#748e;
    unicode[3490]:=16#7490;
    unicode[3491]:=16#749c;
    unicode[3492]:=16#749e;
    unicode[3493]:=16#74a7;
    unicode[3494]:=16#74a8;
    unicode[3495]:=16#74a9;
    unicode[3496]:=16#74ba;
    unicode[3497]:=16#74d2;
    unicode[3498]:=16#74dc;
    unicode[3499]:=16#74de;
    unicode[3500]:=16#74e0;
    unicode[3501]:=16#74e2;
    unicode[3502]:=16#74e3;
    unicode[3503]:=16#74e4;
    unicode[3504]:=16#74e6;
    unicode[3505]:=16#74ee;
    unicode[3506]:=16#74ef;
    unicode[3507]:=16#74f4;
    unicode[3508]:=16#74f6;
    unicode[3509]:=16#74f7;
    unicode[3510]:=16#74ff;
    unicode[3511]:=16#7504;
    unicode[3512]:=16#750d;
    unicode[3513]:=16#750f;
    unicode[3514]:=16#7511;
    unicode[3515]:=16#7513;
    unicode[3516]:=16#7518;
    unicode[3517]:=16#7519;
    unicode[3518]:=16#751a;
    unicode[3519]:=16#751c;
    unicode[3520]:=16#751f;
    unicode[3521]:=16#7525;
    unicode[3522]:=16#7528;
    unicode[3523]:=16#7529;
    unicode[3524]:=16#752b;
    unicode[3525]:=16#752c;
    unicode[3526]:=16#752d;
    unicode[3527]:=16#752f;
    unicode[3528]:=16#7530;
    unicode[3529]:=16#7531;
    unicode[3530]:=16#7532;
    unicode[3531]:=16#7533;
    unicode[3532]:=16#7535;
    unicode[3533]:=16#7537;
    unicode[3534]:=16#7538;
    unicode[3535]:=16#753a;
    unicode[3536]:=16#753b;
    unicode[3537]:=16#753e;
    unicode[3538]:=16#7540;
    unicode[3539]:=16#7545;
    unicode[3540]:=16#7548;
    unicode[3541]:=16#754b;
    unicode[3542]:=16#754c;
    unicode[3543]:=16#754e;
    unicode[3544]:=16#754f;
    unicode[3545]:=16#7554;
    unicode[3546]:=16#7559;
    unicode[3547]:=16#755a;
    unicode[3548]:=16#755b;
    unicode[3549]:=16#755c;
    unicode[3550]:=16#7565;
    unicode[3551]:=16#7566;
    unicode[3552]:=16#756a;
    unicode[3553]:=16#7572;
    unicode[3554]:=16#7574;
    unicode[3555]:=16#7578;
    unicode[3556]:=16#7579;
    unicode[3557]:=16#757f;
    unicode[3558]:=16#7583;
    unicode[3559]:=16#7586;
    unicode[3560]:=16#758b;
    unicode[3561]:=16#758f;
    unicode[3562]:=16#7591;
    unicode[3563]:=16#7592;
    unicode[3564]:=16#7594;
    unicode[3565]:=16#7596;
    unicode[3566]:=16#7597;
    unicode[3567]:=16#7599;
    unicode[3568]:=16#759a;
    unicode[3569]:=16#759d;
    unicode[3570]:=16#759f;
    unicode[3571]:=16#75a0;
    unicode[3572]:=16#75a1;
    unicode[3573]:=16#75a3;
    unicode[3574]:=16#75a4;
    unicode[3575]:=16#75a5;
    unicode[3576]:=16#75ab;
    unicode[3577]:=16#75ac;
    unicode[3578]:=16#75ae;
    unicode[3579]:=16#75af;
    unicode[3580]:=16#75b0;
    unicode[3581]:=16#75b1;
    unicode[3582]:=16#75b2;
    unicode[3583]:=16#75b3;
    unicode[3584]:=16#75b4;
    unicode[3585]:=16#75b5;
    unicode[3586]:=16#75b8;
    unicode[3587]:=16#75b9;
    unicode[3588]:=16#75bc;
    unicode[3589]:=16#75bd;
    unicode[3590]:=16#75be;
    unicode[3591]:=16#75c2;
    unicode[3592]:=16#75c3;
    unicode[3593]:=16#75c4;
    unicode[3594]:=16#75c5;
    unicode[3595]:=16#75c7;
